KUKA KRL program: EPS_2_251719_MHBURNETSTREET_A_20251210010854.src

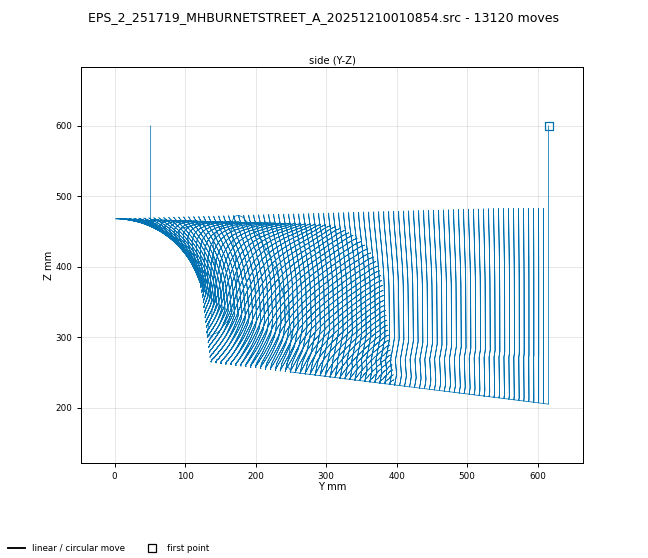
[picture p0: tool path of EPS_2_251719_MHBURNETSTREET_A_20251210010854.src, 13120 of 13122 moves have a stored position in this frame; points joined in program order, loops and branches not executed]
&ACCESS RVP
&REL 4
&COMMENT QRS 19112012
&PARAM EDITMASK = *
DEF PART()
EXT BAS (BAS_COMMAND :IN,REAL :IN )
INT I
BAS (#INITMOV,0 )

;KUKA QRS Post kuka4.cps  Date:22-06-2017 !

File_ID=2951

QRS_PRE_INIT()

;Init var - Until changes are made in qrs_pre_init
Outlet_Square_prg=0
Inlet_1_Square_prg=0
Inlet_2_Square_prg=0
Inlet_3_Square_prg=0
Inlet_4_Square_prg=0
Inlet_5_Square_prg=0

Outlet_1={X 0.000, Y 540.910, Z 382.500, B 0.000, E1 0.000 }
Inlet_1={X 0.000, Y 561.820, Z 357.500, B 0.000, E1 180.000 }
Outlet_1_type=201
Inlet_1_type=0
;QRS#1=Sidecore dimensions
;QRS#2=200-8" PVC SDR 35
;QRS#3=DeadEnd 201
;QRS#4=
;QRS#5=
;QRS#6=
;QRS#7=
;QRS#8=
;QRS#9=12-08 PSX
;QRS#10=

;QRS#11=
;QRS#12=
;QRS#13=
;QRS#14=
;QRS#15=
;QRS#16=1220x127x762 2,5'
;QRS#17=EPS Height
;QRS#18=483
;QRS#19=*
;QRS#20= UPDATED VERSION 22-06-2017
;QRS#21=*
Outlet_Square=0100
Inlet_1_Square=00
Inlet_2_Square=0
Inlet_3_Square=0
Inlet_4_Square=0
Inlet_5_Square=0
Mill_Square=1
Outlet_Square_Prg=204
Inlet_1_Square_prg=0

QRS_INIT()

$ADVANCE=5

; T1
PTP {E1 173.606,E2 173.606}
PTP {X 0,Y 615.507,A -85,B 0,C 180,E1 173.606,E2 173.606,E3 0,E4 0,E5 0,E6 0}
QRS_SPEED_INIT()
LIN {X 0,Y 615.507,Z 600,A -85,B 0,C 180,E1 173.606,E2 173.606,E3 0,E4 0,E5 0,E6 0} C_VEL
LIN {X 0,Y 615.507,Z 215.37,A -85,B 0,C 180,E1 173.606,E2 173.606} C_VEL
LIN {X 0,Y 615.507,Z 207.199,A -85,B 0,C 180,E1 173.606,E2 173.606} C_VEL
LIN {X 0,Y 615.488,Z 205.199,A -85,B 0,C 180,E1 173.42,E2 173.42} C_VEL
LIN {X 0,Y 615.469,Z 205.19,A -85,B 0,C 180,E1 170.801,E2 170.801} C_VEL
LIN {X 0,Y 615.485,Z 205.185,A -85,B 0,C 180,E1 168.14,E2 168.14} C_VEL
LIN {X 0,Y 615.491,Z 205.201,A -85,B 0,C 180,E1 165.451,E2 165.451} C_VEL
LIN {X 0,Y 615.475,Z 205.186,A -85,B 0,C 180,E1 162.73,E2 162.73} C_VEL
LIN {X 0,Y 615.483,Z 205.192,A -85,B 0,C 180,E1 159.968,E2 159.968} C_VEL
LIN {X 0,Y 615.471,Z 205.191,A -85,B 0,C 180,E1 157.155,E2 157.155} C_VEL
LIN {X 0,Y 615.491,Z 205.183,A -85,B 0,C 180,E1 154.43,E2 154.43} C_VEL
LIN {X 0,Y 615.48,Z 205.197,A -85,B 0,C 180,E1 151.551,E2 151.551} C_VEL
LIN {X 0,Y 615.482,Z 205.184,A -85,B 0,C 180,E1 148.915,E2 148.915} C_VEL
LIN {X 0,Y 615.493,Z 205.198,A -85,B 0,C 180,E1 145.979,E2 145.979} C_VEL
LIN {X 0,Y 615.481,Z 205.184,A -85,B 0,C 180,E1 143.064,E2 143.064} C_VEL
LIN {X 0,Y 615.482,Z 205.195,A -85,B 0,C 180,E1 140.25,E2 140.25} C_VEL
LIN {X 0,Y 615.475,Z 205.193,A -85,B 0,C 180,E1 137.647,E2 137.647} C_VEL
LIN {X 0,Y 615.495,Z 205.181,A -85,B 0,C 180,E1 134.933,E2 134.933} C_VEL
LIN {X 0,Y 615.493,Z 205.199,A -85,B 0,C 180,E1 132.081,E2 132.081} C_VEL
LIN {X 0,Y 615.473,Z 205.192,A -85,B 0,C 180,E1 129.751,E2 129.751} C_VEL
LIN {X 0,Y 615.485,Z 205.185,A -85,B 0,C 180,E1 126.937,E2 126.937} C_VEL
LIN {X 0,Y 615.48,Z 205.195,A -85,B 0,C 180,E1 124.022,E2 124.022} C_VEL
LIN {X 0,Y 615.474,Z 205.188,A -85,B 0,C 180,E1 121.686,E2 121.686} C_VEL
LIN {X 0,Y 615.487,Z 205.183,A -85,B 0,C 180,E1 119.406,E2 119.406} C_VEL
LIN {X 0,Y 615.49,Z 205.201,A -85,B 0,C 180,E1 116.444,E2 116.444} C_VEL
LIN {X 0,Y 615.486,Z 205.183,A -85,B 0,C 180,E1 113.556,E2 113.556} C_VEL
LIN {X 0,Y 615.485,Z 205.198,A -85,B 0,C 180,E1 110.731,E2 110.731} C_VEL
LIN {X 0,Y 615.478,Z 205.187,A -85,B 0,C 180,E1 107.957,E2 107.957} C_VEL
LIN {X 0,Y 615.479,Z 205.189,A -85,B 0,C 180,E1 105.226,E2 105.226} C_VEL
LIN {X 0,Y 615.484,Z 205.196,A -85,B 0,C 180,E1 102.53,E2 102.53} C_VEL
LIN {X 0,Y 615.493,Z 205.181,A -85,B 0,C 180,E1 99.862,E2 99.862} C_VEL
LIN {X 0,Y 615.48,Z 205.193,A -85,B 0,C 180,E1 97.216,E2 97.216} C_VEL
LIN {X 0,Y 615.48,Z 205.194,A -85,B 0,C 180,E1 94.585,E2 94.585} C_VEL
LIN {X 0,Y 615.5,Z 205.18,A -85,B 0,C 180,E1 91.963,E2 91.963} C_VEL
LIN {X 0,Y 615.48,Z 205.193,A -85,B 0,C 180,E1 89.346,E2 89.346} C_VEL
LIN {X 0,Y 615.48,Z 205.193,A -85,B 0,C 180,E1 86.727,E2 86.727} C_VEL
LIN {X 0,Y 615.498,Z 205.18,A -85,B 0,C 180,E1 84.102,E2 84.102} C_VEL
LIN {X 0,Y 615.481,Z 205.194,A -85,B 0,C 180,E1 81.463,E2 81.463} C_VEL
LIN {X 0,Y 615.477,Z 205.192,A -85,B 0,C 180,E1 78.807,E2 78.807} C_VEL
LIN {X 0,Y 615.483,Z 205.184,A -85,B 0,C 180,E1 76.067,E2 76.067} C_VEL
LIN {X 0,Y 615.493,Z 205.199,A -85,B 0,C 180,E1 73.414,E2 73.414} C_VEL
LIN {X 0,Y 615.485,Z 205.185,A -85,B 0,C 180,E1 70.662,E2 70.662} C_VEL
LIN {X 0,Y 615.477,Z 205.192,A -85,B 0,C 180,E1 67.863,E2 67.863} C_VEL
LIN {X 0,Y 615.48,Z 205.19,A -85,B 0,C 180,E1 65.008,E2 65.008} C_VEL
LIN {X 0,Y 615.484,Z 205.185,A -85,B 0,C 180,E1 62.823,E2 62.823} C_VEL
LIN {X 0,Y 615.475,Z 205.188,A -85,B 0,C 180,E1 60.206,E2 60.206} C_VEL
LIN {X 0,Y 615.492,Z 205.198,A -85,B 0,C 180,E1 57.543,E2 57.543} C_VEL
LIN {X 0,Y 615.481,Z 205.189,A -85,B 0,C 180,E1 55.185,E2 55.185} C_VEL
LIN {X 0,Y 615.492,Z 205.182,A -85,B 0,C 180,E1 52.758,E2 52.758} C_VEL
LIN {X 0,Y 615.491,Z 205.198,A -85,B 0,C 180,E1 49.91,E2 49.91} C_VEL
LIN {X 0,Y 615.488,Z 205.183,A -85,B 0,C 180,E1 46.952,E2 46.952} C_VEL
LIN {X 0,Y 615.482,Z 205.196,A -85,B 0,C 180,E1 44.149,E2 44.149} C_VEL
LIN {X 0,Y 615.482,Z 205.189,A -85,B 0,C 180,E1 41.474,E2 41.474} C_VEL
LIN {X 0,Y 615.482,Z 205.184,A -85,B 0,C 180,E1 38.904,E2 38.904} C_VEL
LIN {X 0,Y 615.476,Z 205.194,A -85,B 0,C 180,E1 36.425,E2 36.425} C_VEL
LIN {X 0,Y 615.485,Z 205.186,A -85,B 0,C 180,E1 33.534,E2 33.534} C_VEL
LIN {X 0,Y 615.474,Z 205.187,A -85,B 0,C 180,E1 30.92,E2 30.92} C_VEL
LIN {X 0,Y 615.48,Z 205.197,A -85,B 0,C 180,E1 28.449,E2 28.449} C_VEL
LIN {X 0,Y 615.487,Z 205.184,A -85,B 0,C 180,E1 25.569,E2 25.569} C_VEL
LIN {X 0,Y 615.471,Z 205.191,A -85,B 0,C 180,E1 22.845,E2 22.845} C_VEL
LIN {X 0,Y 615.486,Z 205.197,A -85,B 0,C 180,E1 20.557,E2 20.557} C_VEL
LIN {X 0,Y 615.484,Z 205.189,A -85,B 0,C 180,E1 17.957,E2 17.957} C_VEL
LIN {X 0,Y 615.472,Z 205.188,A -85,B 0,C 180,E1 15.226,E2 15.226} C_VEL
LIN {X 0,Y 615.489,Z 205.202,A -85,B 0,C 180,E1 12.53,E2 12.53} C_VEL
LIN {X 0,Y 615.495,Z 205.182,A -85,B 0,C 180,E1 9.862,E2 9.862} C_VEL
LIN {X 0,Y 615.469,Z 205.191,A -85,B 0,C 180,E1 7.215,E2 7.215} C_VEL
LIN {X 0,Y 615.492,Z 205.197,A -85,B 0,C 180,E1 4.584,E2 4.584} C_VEL
LIN {X 0,Y 615.5,Z 205.181,A -85,B 0,C 180,E1 1.963,E2 1.963} C_VEL
LIN {X 0,Y 615.468,Z 205.191,A -85,B 0,C 180,E1 -0.655,E2 -0.655} C_VEL
LIN {X 0,Y 615.492,Z 205.197,A -85,B 0,C 180,E1 -3.273,E2 -3.273} C_VEL
LIN {X 0,Y 615.497,Z 205.181,A -85,B 0,C 180,E1 -5.899,E2 -5.899} C_VEL
LIN {X 0,Y 615.468,Z 205.192,A -85,B 0,C 180,E1 -8.537,E2 -8.537} C_VEL
LIN {X 0,Y 615.489,Z 205.195,A -85,B 0,C 180,E1 -11.193,E2 -11.193} C_VEL
LIN {X 0,Y 615.479,Z 205.184,A -85,B 0,C 180,E1 -13.93,E2 -13.93} C_VEL
LIN {X 0,Y 615.476,Z 205.196,A -85,B 0,C 180,E1 -16.587,E2 -16.587} C_VEL
LIN {X 0,Y 615.489,Z 205.187,A -85,B 0,C 180,E1 -19.338,E2 -19.338} C_VEL
LIN {X 0,Y 615.465,Z 205.191,A -85,B 0,C 180,E1 -22.138,E2 -22.138} C_VEL
LIN {X 0,Y 615.488,Z 205.193,A -85,B 0,C 180,E1 -24.992,E2 -24.992} C_VEL
LIN {X 0,Y 615.466,Z 205.189,A -85,B 0,C 180,E1 -27.916,E2 -27.916} C_VEL
LIN {X 0,Y 615.468,Z 205.194,A -85,B 0,C 180,E1 -30.161,E2 -30.161} C_VEL
LIN {X 0,Y 615.487,Z 205.2,A -85,B 0,C 180,E1 -32.458,E2 -32.458} C_VEL
LIN {X 0,Y 615.488,Z 205.192,A -85,B 0,C 180,E1 -34.815,E2 -34.815} C_VEL
LIN {X 0,Y 615.49,Z 205.183,A -85,B 0,C 180,E1 -37.242,E2 -37.242} C_VEL
LIN {X 0,Y 615.472,Z 205.196,A -85,B 0,C 180,E1 -40.088,E2 -40.088} C_VEL
LIN {X 0,Y 615.488,Z 205.184,A -85,B 0,C 180,E1 -43.048,E2 -43.048} C_VEL
LIN {X 0,Y 615.467,Z 205.194,A -85,B 0,C 180,E1 -45.849,E2 -45.849} C_VEL
LIN {X 0,Y 615.489,Z 205.192,A -85,B 0,C 180,E1 -48.527,E2 -48.527} C_VEL
LIN {X 0,Y 615.478,Z 205.185,A -85,B 0,C 180,E1 -51.095,E2 -51.095} C_VEL
LIN {X 0,Y 615.463,Z 205.192,A -85,B 0,C 180,E1 -53.574,E2 -53.574} C_VEL
LIN {X 0,Y 615.49,Z 205.189,A -85,B 0,C 180,E1 -56.466,E2 -56.466} C_VEL
LIN {X 0,Y 615.467,Z 205.187,A -85,B 0,C 180,E1 -59.079,E2 -59.079} C_VEL
LIN {X 0,Y 615.466,Z 205.195,A -85,B 0,C 180,E1 -61.554,E2 -61.554} C_VEL
LIN {X 0,Y 615.49,Z 205.187,A -85,B 0,C 180,E1 -64.431,E2 -64.431} C_VEL
LIN {X 0,Y 615.497,Z 205.361,A -85,B 0,C 180,E1 -65.958,E2 -65.958} C_VEL
LIN {X 0,Y 615.49,Z 220.439,A -85,B 0,C 180,E1 -68.568,E2 -68.568} C_VEL
LIN {X 0,Y 615.483,Z 237.22,A -85,B 0,C 180,E1 -71.397,E2 -71.397} C_VEL
LIN {X 0,Y 615.498,Z 254.497,A -85,B 0,C 180,E1 -74.265,E2 -74.265} C_VEL
LIN {X 0,Y 615.469,Z 271.731,A -85,B 0,C 180,E1 -77.071,E2 -77.071} C_VEL
LIN {X 0,Y 615.463,Z 273.25,A -85,B 0,C 180,E1 -77.155,E2 -77.155} C_VEL
LIN {X 0,Y 615.498,Z 378.83,A -85,B 0,C 180,E1 -78.411,E2 -78.411} C_VEL
LIN {X 0,Y 615.499,Z 391.343,A -85,B 0,C 180,E1 -78.682,E2 -78.682} C_VEL
LIN {X 0,Y 615.496,Z 404.502,A -85,B 0,C 180,E1 -79.109,E2 -79.109} C_VEL
LIN {X 0,Y 615.488,Z 416.478,A -85,B 0,C 180,E1 -79.639,E2 -79.639} C_VEL
LIN {X 0,Y 615.494,Z 427.994,A -85,B 0,C 180,E1 -80.304,E2 -80.304} C_VEL
LIN {X 0,Y 615.499,Z 438.341,A -85,B 0,C 180,E1 -81.05,E2 -81.05} C_VEL
LIN {X 0,Y 615.497,Z 446.812,A -85,B 0,C 180,E1 -81.794,E2 -81.794} C_VEL
LIN {X 0,Y 615.498,Z 454.606,A -85,B 0,C 180,E1 -82.62,E2 -82.62} C_VEL
LIN {X 0,Y 615.496,Z 462.203,A -85,B 0,C 180,E1 -83.608,E2 -83.608} C_VEL
LIN {X 0,Y 615.498,Z 469.205,A -85,B 0,C 180,E1 -84.759,E2 -84.759} C_VEL
LIN {X 0,Y 615.494,Z 473.851,A -85,B 0,C 180,E1 -85.744,E2 -85.744} C_VEL
LIN {X 0,Y 615.494,Z 477.399,A -85,B 0,C 180,E1 -86.727,E2 -86.727} C_VEL
LIN {X 0,Y 615.497,Z 479.233,A -85,B 0,C 180,E1 -87.382,E2 -87.382} C_VEL
LIN {X 0,Y 615.5,Z 480.607,A -85,B 0,C 180,E1 -88.037,E2 -88.037} C_VEL
LIN {X 0,Y 615.496,Z 482.173,A -85,B 0,C 180,E1 -89.346,E2 -89.346} C_VEL
LIN {X 0,Y 615.494,Z 482.389,A -85,B 0,C 180,E1 -90,E2 -90} C_VEL
LIN {X 0,Y 615.495,Z 481.58,A -85,B 0,C 180,E1 -91.309,E2 -91.309} C_VEL
LIN {X 0,Y 615.5,Z 480.607,A -85,B 0,C 180,E1 -91.963,E2 -91.963} C_VEL
LIN {X 0,Y 615.497,Z 479.233,A -85,B 0,C 180,E1 -92.618,E2 -92.618} C_VEL
LIN {X 0,Y 615.496,Z 476.349,A -85,B 0,C 180,E1 -93.601,E2 -93.601} C_VEL
LIN {X 0,Y 615.498,Z 472.441,A -85,B 0,C 180,E1 -94.584,E2 -94.584} C_VEL
LIN {X 0,Y 615.499,Z 467.405,A -85,B 0,C 180,E1 -95.57,E2 -95.57} C_VEL
LIN {X 0,Y 615.497,Z 460.87,A -85,B 0,C 180,E1 -96.583,E2 -96.583} C_VEL
LIN {X 0,Y 615.497,Z 453.133,A -85,B 0,C 180,E1 -97.545,E2 -97.545} C_VEL
LIN {X 0,Y 615.498,Z 445.045,A -85,B 0,C 180,E1 -98.371,E2 -98.371} C_VEL
LIN {X 0,Y 615.499,Z 435.168,A -85,B 0,C 180,E1 -99.199,E2 -99.199} C_VEL
LIN {X 0,Y 615.491,Z 423.982,A -85,B 0,C 180,E1 -99.945,E2 -99.945} C_VEL
LIN {X 0,Y 615.493,Z 413.022,A -85,B 0,C 180,E1 -100.527,E2 -100.527} C_VEL
LIN {X 0,Y 615.499,Z 400.419,A -85,B 0,C 180,E1 -101.042,E2 -101.042} C_VEL
LIN {X 0,Y 615.499,Z 388.065,A -85,B 0,C 180,E1 -101.401,E2 -101.401} C_VEL
LIN {X 0,Y 615.499,Z 374.466,A -85,B 0,C 180,E1 -101.652,E2 -101.652} C_VEL
LIN {X 0,Y 615.465,Z 272.546,A -85,B 0,C 180,E1 -102.866,E2 -102.866} C_VEL
LIN {X 0,Y 615.478,Z 270.987,A -85,B 0,C 180,E1 -103.033,E2 -103.033} C_VEL
LIN {X 0,Y 615.494,Z 253.464,A -85,B 0,C 180,E1 -105.905,E2 -105.905} C_VEL
LIN {X 0,Y 615.484,Z 236.96,A -85,B 0,C 180,E1 -108.646,E2 -108.646} C_VEL
LIN {X 0,Y 615.49,Z 220.439,A -85,B 0,C 180,E1 -111.432,E2 -111.432} C_VEL
LIN {X 0,Y 615.497,Z 205.361,A -85,B 0,C 180,E1 -114.042,E2 -114.042} C_VEL
LIN {X 0,Y 615.468,Z 205.195,A -85,B 0,C 180,E1 -116.445,E2 -116.445} C_VEL
LIN {X 0,Y 615.461,Z 205.192,A -85,B 0,C 180,E1 -118.659,E2 -118.659} C_VEL
LIN {X 0,Y 615.478,Z 205.185,A -85,B 0,C 180,E1 -121.084,E2 -121.084} C_VEL
LIN {X 0,Y 615.486,Z 205.2,A -85,B 0,C 180,E1 -124.022,E2 -124.022} C_VEL
LIN {X 0,Y 615.463,Z 205.192,A -85,B 0,C 180,E1 -126.426,E2 -126.426} C_VEL
LIN {X 0,Y 615.493,Z 205.183,A -85,B 0,C 180,E1 -129.062,E2 -129.062} C_VEL
LIN {X 0,Y 615.472,Z 205.196,A -85,B 0,C 180,E1 -132.078,E2 -132.078} C_VEL
LIN {X 0,Y 615.493,Z 205.182,A -85,B 0,C 180,E1 -134.932,E2 -134.932} C_VEL
LIN {X 0,Y 615.475,Z 205.196,A -85,B 0,C 180,E1 -137.921,E2 -137.921} C_VEL
LIN {X 0,Y 615.462,Z 205.191,A -85,B 0,C 180,E1 -140.248,E2 -140.248} C_VEL
LIN {X 0,Y 615.49,Z 205.188,A -85,B 0,C 180,E1 -143.063,E2 -143.063} C_VEL
LIN {X 0,Y 615.466,Z 205.193,A -85,B 0,C 180,E1 -145.976,E2 -145.976} C_VEL
LIN {X 0,Y 615.467,Z 205.188,A -85,B 0,C 180,E1 -148.313,E2 -148.313} C_VEL
LIN {X 0,Y 615.486,Z 205.184,A -85,B 0,C 180,E1 -150.593,E2 -150.593} C_VEL
LIN {X 0,Y 615.478,Z 205.197,A -85,B 0,C 180,E1 -153.555,E2 -153.555} C_VEL
LIN {X 0,Y 615.465,Z 205.189,A -85,B 0,C 180,E1 -155.996,E2 -155.996} C_VEL
LIN {X 0,Y 615.495,Z 205.183,A -85,B 0,C 180,E1 -158.568,E2 -158.568} C_VEL
LIN {X 0,Y 615.479,Z 205.197,A -85,B 0,C 180,E1 -161.397,E2 -161.397} C_VEL
LIN {X 0,Y 615.478,Z 205.185,A -85,B 0,C 180,E1 -164.094,E2 -164.094} C_VEL
LIN {X 0,Y 615.486,Z 205.194,A -85,B 0,C 180,E1 -166.798,E2 -166.798} C_VEL
LIN {X 0,Y 615.469,Z 205.193,A -85,B 0,C 180,E1 -169.472,E2 -169.472} C_VEL
LIN {X 0,Y 615.485,Z 205.184,A -85,B 0,C 180,E1 -172.124,E2 -172.124} C_VEL
LIN {X 0,Y 615.489,Z 205.197,A -85,B 0,C 180,E1 -174.758,E2 -174.758} C_VEL
LIN {X 0,Y 615.465,Z 205.192,A -85,B 0,C 180,E1 -177.382,E2 -177.382} C_VEL
LIN {X 0,Y 615.486,Z 205.184,A -85,B 0,C 180,E1 -180,E2 -180} C_VEL
LIN {X 0,Y 615.488,Z 205.198,A -85,B 0,C 180,E1 -182.617,E2 -182.617} C_VEL
LIN {X 0,Y 615.468,Z 205.191,A -85,B 0,C 180,E1 -185.241,E2 -185.241} C_VEL
LIN {X 0,Y 615.488,Z 205.199,A -85,B 0,C 180,E1 -186.58,E2 -186.58} C_VEL
LIN {X 0,Y 614.798,Z 205.338,A -85,B 0,C 180,E1 -187.126,E2 -187.126} C_VEL
LIN {X 0,Y 611.952,Z 205.753,A -85,B 0,C 180,E1 -188.012,E2 -188.012} C_VEL
LIN {X 0,Y 609.562,Z 206.062,A -85,B 0,C 180,E1 -188.725,E2 -188.725} C_VEL
LIN {X 0,Y 608.536,Z 206.179,A -85,B 0,C 180,E1 -189.274,E2 -189.274} C_VEL
LIN {X 0,Y 608.452,Z 206.187,A -85,B 0,C 180,E1 -189.46,E2 -189.46} C_VEL
LIN {X 0,Y 608.462,Z 206.188,A -85,B 0,C 180,E1 -191.999,E2 -191.999} C_VEL
LIN {X 0,Y 608.474,Z 206.192,A -85,B 0,C 180,E1 -194.72,E2 -194.72} C_VEL
LIN {X 0,Y 608.445,Z 206.188,A -85,B 0,C 180,E1 -197.476,E2 -197.476} C_VEL
LIN {X 0,Y 608.461,Z 206.194,A -85,B 0,C 180,E1 -200.274,E2 -200.274} C_VEL
LIN {X 0,Y 608.456,Z 206.196,A -85,B 0,C 180,E1 -202.476,E2 -202.476} C_VEL
LIN {X 0,Y 608.449,Z 206.194,A -85,B 0,C 180,E1 -204.571,E2 -204.571} C_VEL
LIN {X 0,Y 608.473,Z 206.185,A -85,B 0,C 180,E1 -207.207,E2 -207.207} C_VEL
LIN {X 0,Y 608.469,Z 206.192,A -85,B 0,C 180,E1 -209.972,E2 -209.972} C_VEL
LIN {X 0,Y 608.454,Z 206.192,A -85,B 0,C 180,E1 -212.522,E2 -212.522} C_VEL
LIN {X 0,Y 608.44,Z 206.189,A -85,B 0,C 180,E1 -214.905,E2 -214.905} C_VEL
LIN {X 0,Y 608.479,Z 206.184,A -85,B 0,C 180,E1 -217.16,E2 -217.16} C_VEL
LIN {X 0,Y 608.474,Z 206.187,A -85,B 0,C 180,E1 -219.439,E2 -219.439} C_VEL
LIN {X 0,Y 608.447,Z 206.192,A -85,B 0,C 180,E1 -222.333,E2 -222.333} C_VEL
LIN {X 0,Y 608.46,Z 206.187,A -85,B 0,C 180,E1 -224.795,E2 -224.795} C_VEL
LIN {X 0,Y 608.454,Z 206.187,A -85,B 0,C 180,E1 -227.04,E2 -227.04} C_VEL
LIN {X 0,Y 608.453,Z 206.196,A -85,B 0,C 180,E1 -229.697,E2 -229.697} C_VEL
LIN {X 0,Y 608.469,Z 206.188,A -85,B 0,C 180,E1 -232.254,E2 -232.254} C_VEL
LIN {X 0,Y 608.445,Z 206.19,A -85,B 0,C 180,E1 -235.094,E2 -235.094} C_VEL
LIN {X 0,Y 608.467,Z 206.192,A -85,B 0,C 180,E1 -237.906,E2 -237.906} C_VEL
LIN {X 0,Y 608.46,Z 206.188,A -85,B 0,C 180,E1 -240.22,E2 -240.22} C_VEL
LIN {X 0,Y 608.477,Z 206.185,A -85,B 0,C 180,E1 -242.792,E2 -242.792} C_VEL
LIN {X 0,Y 608.449,Z 206.198,A -85,B 0,C 180,E1 -245.429,E2 -245.429} C_VEL
LIN {X 0,Y 608.469,Z 206.186,A -85,B 0,C 180,E1 -248.309,E2 -248.309} C_VEL
LIN {X 0,Y 608.472,Z 206.194,A -85,B 0,C 180,E1 -251.282,E2 -251.282} C_VEL
LIN {X 0,Y 608.457,Z 206.189,A -85,B 0,C 180,E1 -253.906,E2 -253.906} C_VEL
LIN {X 0,Y 608.459,Z 206.188,A -85,B 0,C 180,E1 -256.644,E2 -256.644} C_VEL
LIN {X 0,Y 608.463,Z 206.194,A -85,B 0,C 180,E1 -259.35,E2 -259.35} C_VEL
LIN {X 0,Y 608.477,Z 206.185,A -85,B 0,C 180,E1 -262.033,E2 -262.033} C_VEL
LIN {X 0,Y 608.461,Z 206.19,A -85,B 0,C 180,E1 -264.698,E2 -264.698} C_VEL
LIN {X 0,Y 608.472,Z 206.191,A -85,B 0,C 180,E1 -267.352,E2 -267.352} C_VEL
LIN {X 0,Y 608.477,Z 206.185,A -85,B 0,C 180,E1 -270,E2 -270} C_VEL
LIN {X 0,Y 608.472,Z 206.191,A -85,B 0,C 180,E1 -272.648,E2 -272.648} C_VEL
LIN {X 0,Y 608.461,Z 206.19,A -85,B 0,C 180,E1 -275.302,E2 -275.302} C_VEL
LIN {X 0,Y 608.477,Z 206.185,A -85,B 0,C 180,E1 -277.967,E2 -277.967} C_VEL
LIN {X 0,Y 608.468,Z 206.193,A -85,B 0,C 180,E1 -280.958,E2 -280.958} C_VEL
LIN {X 0,Y 608.459,Z 206.188,A -85,B 0,C 180,E1 -283.356,E2 -283.356} C_VEL
LIN {X 0,Y 608.457,Z 206.189,A -85,B 0,C 180,E1 -286.094,E2 -286.094} C_VEL
LIN {X 0,Y 608.456,Z 206.193,A -85,B 0,C 180,E1 -288.87,E2 -288.87} C_VEL
LIN {X 0,Y 608.469,Z 206.186,A -85,B 0,C 180,E1 -291.691,E2 -291.691} C_VEL
LIN {X 0,Y 608.449,Z 206.198,A -85,B 0,C 180,E1 -294.571,E2 -294.571} C_VEL
LIN {X 0,Y 608.477,Z 206.185,A -85,B 0,C 180,E1 -297.208,E2 -297.208} C_VEL
LIN {X 0,Y 608.458,Z 206.19,A -85,B 0,C 180,E1 -299.971,E2 -299.971} C_VEL
LIN {X 0,Y 608.466,Z 206.193,A -85,B 0,C 180,E1 -302.524,E2 -302.524} C_VEL
LIN {X 0,Y 608.435,Z 206.189,A -85,B 0,C 180,E1 -305.278,E2 -305.278} C_VEL
LIN {X 0,Y 608.469,Z 206.188,A -85,B 0,C 180,E1 -307.746,E2 -307.746} C_VEL
LIN {X 0,Y 608.452,Z 206.195,A -85,B 0,C 180,E1 -310.33,E2 -310.33} C_VEL
LIN {X 0,Y 608.454,Z 206.187,A -85,B 0,C 180,E1 -312.96,E2 -312.96} C_VEL
LIN {X 0,Y 608.453,Z 206.192,A -85,B 0,C 180,E1 -315.736,E2 -315.736} C_VEL
LIN {X 0,Y 608.46,Z 206.188,A -85,B 0,C 180,E1 -318.658,E2 -318.658} C_VEL
LIN {X 0,Y 608.466,Z 206.188,A -85,B 0,C 180,E1 -321.412,E2 -321.412} C_VEL
LIN {X 0,Y 608.474,Z 206.195,A -85,B 0,C 180,E1 -323.951,E2 -323.951} C_VEL
LIN {X 0,Y 608.465,Z 206.189,A -85,B 0,C 180,E1 -326.33,E2 -326.33} C_VEL
LIN {X 0,Y 608.474,Z 206.185,A -85,B 0,C 180,E1 -328.728,E2 -328.728} C_VEL
LIN {X 0,Y 608.464,Z 206.19,A -85,B 0,C 180,E1 -331.381,E2 -331.381} C_VEL
LIN {X 0,Y 608.443,Z 206.195,A -85,B 0,C 180,E1 -333.965,E2 -333.965} C_VEL
LIN {X 0,Y 608.466,Z 206.189,A -85,B 0,C 180,E1 -336.156,E2 -336.156} C_VEL
LIN {X 0,Y 608.472,Z 206.186,A -85,B 0,C 180,E1 -338.309,E2 -338.309} C_VEL
LIN {X 0,Y 608.468,Z 206.191,A -85,B 0,C 180,E1 -341.284,E2 -341.284} C_VEL
LIN {X 0,Y 608.462,Z 206.19,A -85,B 0,C 180,E1 -343.907,E2 -343.907} C_VEL
LIN {X 0,Y 608.453,Z 206.188,A -85,B 0,C 180,E1 -346.644,E2 -346.644} C_VEL
LIN {X 0,Y 608.463,Z 206.196,A -85,B 0,C 180,E1 -349.351,E2 -349.351} C_VEL
LIN {X 0,Y 608.479,Z 206.185,A -85,B 0,C 180,E1 -352.033,E2 -352.033} C_VEL
LIN {X 0,Y 608.45,Z 206.189,A -85,B 0,C 180,E1 -354.698,E2 -354.698} C_VEL
LIN {X 0,Y 608.478,Z 206.193,A -85,B 0,C 180,E1 -357.352,E2 -357.352} C_VEL
LIN {X 0,Y 608.477,Z 206.184,A -85,B 0,C 180,E1 -360,E2 -360} C_VEL
LIN {X 0,Y 608.459,Z 206.189,A -85,B 0,C 180,E1 -362.648,E2 -362.648} C_VEL
LIN {X 0,Y 608.469,Z 206.192,A -85,B 0,C 180,E1 -365.302,E2 -365.302} C_VEL
LIN {X 0,Y 608.475,Z 206.184,A -85,B 0,C 180,E1 -367.967,E2 -367.967} C_VEL
LIN {X 0,Y 608.453,Z 206.192,A -85,B 0,C 180,E1 -370.65,E2 -370.65} C_VEL
LIN {X 0,Y 608.463,Z 206.19,A -85,B 0,C 180,E1 -373.357,E2 -373.357} C_VEL
LIN {X 0,Y 608.45,Z 206.188,A -85,B 0,C 180,E1 -376.094,E2 -376.094} C_VEL
LIN {X 0,Y 608.453,Z 206.197,A -85,B 0,C 180,E1 -378.87,E2 -378.87} C_VEL
LIN {X 0,Y 608.466,Z 206.186,A -85,B 0,C 180,E1 -381.692,E2 -381.692} C_VEL
LIN {X 0,Y 608.445,Z 206.197,A -85,B 0,C 180,E1 -384.572,E2 -384.572} C_VEL
LIN {X 0,Y 608.481,Z 206.186,A -85,B 0,C 180,E1 -387.208,E2 -387.208} C_VEL
LIN {X 0,Y 608.451,Z 206.189,A -85,B 0,C 180,E1 -389.969,E2 -389.969} C_VEL
LIN {X 0,Y 608.459,Z 206.191,A -85,B 0,C 180,E1 -392.88,E2 -392.88} C_VEL
LIN {X 0,Y 608.435,Z 206.19,A -85,B 0,C 180,E1 -395.279,E2 -395.279} C_VEL
LIN {X 0,Y 608.459,Z 206.188,A -85,B 0,C 180,E1 -397.747,E2 -397.747} C_VEL
LIN {X 0,Y 608.446,Z 206.198,A -85,B 0,C 180,E1 -400.329,E2 -400.329} C_VEL
LIN {X 0,Y 608.469,Z 206.185,A -85,B 0,C 180,E1 -403.309,E2 -403.309} C_VEL
LIN {X 0,Y 608.463,Z 206.194,A -85,B 0,C 180,E1 -406.13,E2 -406.13} C_VEL
LIN {X 0,Y 608.457,Z 206.188,A -85,B 0,C 180,E1 -408.824,E2 -408.824} C_VEL
LIN {X 0,Y 608.433,Z 206.19,A -85,B 0,C 180,E1 -411.41,E2 -411.41} C_VEL
LIN {X 0,Y 608.448,Z 206.196,A -85,B 0,C 180,E1 -413.955,E2 -413.955} C_VEL
LIN {X 0,Y 608.466,Z 206.192,A -85,B 0,C 180,E1 -416.33,E2 -416.33} C_VEL
LIN {X 0,Y 608.447,Z 206.189,A -85,B 0,C 180,E1 -418.733,E2 -418.733} C_VEL
LIN {X 0,Y 608.454,Z 206.189,A -85,B 0,C 180,E1 -421.384,E2 -421.384} C_VEL
LIN {X 0,Y 608.439,Z 206.2,A -85,B 0,C 180,E1 -423.964,E2 -423.964} C_VEL
LIN {X 0,Y 608.496,Z 206.349,A -85,B 0,C 180,E1 -425.844,E2 -425.844} C_VEL
LIN {X 0,Y 608.529,Z 220.462,A -85,B 0,C 180,E1 -428.311,E2 -428.311} C_VEL
LIN {X 0,Y 608.51,Z 237.019,A -85,B 0,C 180,E1 -431.132,E2 -431.132} C_VEL
LIN {X 0,Y 608.483,Z 253.576,A -85,B 0,C 180,E1 -433.907,E2 -433.907} C_VEL
LIN {X 0,Y 608.48,Z 270.133,A -85,B 0,C 180,E1 -436.644,E2 -436.644} C_VEL
LIN {X 0,Y 608.461,Z 272.248,A -85,B 0,C 180,E1 -436.962,E2 -436.962} C_VEL
LIN {X 0,Y 608.539,Z 274.724,A -85,B 0,C 180,E1 -437.028,E2 -437.028} C_VEL
LIN {X 0,Y 608.548,Z 378.941,A -85,B 0,C 180,E1 -438.277,E2 -438.277} C_VEL
LIN {X 0,Y 608.548,Z 392.226,A -85,B 0,C 180,E1 -438.572,E2 -438.572} C_VEL
LIN {X 0,Y 608.54,Z 405.391,A -85,B 0,C 180,E1 -439.011,E2 -439.011} C_VEL
LIN {X 0,Y 608.51,Z 416.623,A -85,B 0,C 180,E1 -439.519,E2 -439.519} C_VEL
LIN {X 0,Y 608.485,Z 428.198,A -85,B 0,C 180,E1 -440.191,E2 -440.191} C_VEL
LIN {X 0,Y 608.485,Z 438.596,A -85,B 0,C 180,E1 -440.946,E2 -440.946} C_VEL
LIN {X 0,Y 608.475,Z 447.114,A -85,B 0,C 180,E1 -441.699,E2 -441.699} C_VEL
LIN {X 0,Y 608.471,Z 454.959,A -85,B 0,C 180,E1 -442.534,E2 -442.534} C_VEL
LIN {X 0,Y 608.461,Z 462.286,A -85,B 0,C 180,E1 -443.485,E2 -443.485} C_VEL
LIN {X 0,Y 608.451,Z 467.864,A -85,B 0,C 180,E1 -444.366,E2 -444.366} C_VEL
LIN {X 0,Y 608.432,Z 472.95,A -85,B 0,C 180,E1 -445.362,E2 -445.362} C_VEL
LIN {X 0,Y 608.449,Z 476.896,A -85,B 0,C 180,E1 -446.358,E2 -446.358} C_VEL
LIN {X 0,Y 608.425,Z 479.808,A -85,B 0,C 180,E1 -447.352,E2 -447.352} C_VEL
LIN {X 0,Y 608.445,Z 481.201,A -85,B 0,C 180,E1 -448.014,E2 -448.014} C_VEL
LIN {X 0,Y 608.438,Z 482.783,A -85,B 0,C 180,E1 -449.338,E2 -449.338} C_VEL
LIN {X 0,Y 608.434,Z 482.998,A -85,B 0,C 180,E1 -450,E2 -450} C_VEL
LIN {X 0,Y 608.448,Z 482.184,A -85,B 0,C 180,E1 -451.324,E2 -451.324} C_VEL
LIN {X 0,Y 608.445,Z 481.201,A -85,B 0,C 180,E1 -451.986,E2 -451.986} C_VEL
LIN {X 0,Y 608.425,Z 479.808,A -85,B 0,C 180,E1 -452.648,E2 -452.648} C_VEL
LIN {X 0,Y 608.449,Z 476.896,A -85,B 0,C 180,E1 -453.642,E2 -453.642} C_VEL
LIN {X 0,Y 608.432,Z 472.95,A -85,B 0,C 180,E1 -454.638,E2 -454.638} C_VEL
LIN {X 0,Y 608.451,Z 467.864,A -85,B 0,C 180,E1 -455.634,E2 -455.634} C_VEL
LIN {X 0,Y 608.442,Z 461.472,A -85,B 0,C 180,E1 -456.633,E2 -456.633} C_VEL
LIN {X 0,Y 608.475,Z 453.479,A -85,B 0,C 180,E1 -457.633,E2 -457.633} C_VEL
LIN {X 0,Y 608.487,Z 445.338,A -85,B 0,C 180,E1 -458.468,E2 -458.468} C_VEL
LIN {X 0,Y 608.487,Z 435.396,A -85,B 0,C 180,E1 -459.306,E2 -459.306} C_VEL
LIN {X 0,Y 608.505,Z 424.168,A -85,B 0,C 180,E1 -460.06,E2 -460.06} C_VEL
LIN {X 0,Y 608.518,Z 413.176,A -85,B 0,C 180,E1 -460.649,E2 -460.649} C_VEL
LIN {X 0,Y 608.535,Z 401.706,A -85,B 0,C 180,E1 -461.127,E2 -461.127} C_VEL
LIN {X 0,Y 608.55,Z 389.069,A -85,B 0,C 180,E1 -461.512,E2 -461.512} C_VEL
LIN {X 0,Y 608.563,Z 376.111,A -85,B 0,C 180,E1 -461.765,E2 -461.765} C_VEL
LIN {X 0,Y 608.48,Z 272.577,A -85,B 0,C 180,E1 -463.016,E2 -463.016} C_VEL
LIN {X 0,Y 608.456,Z 271.167,A -85,B 0,C 180,E1 -463.187,E2 -463.187} C_VEL
LIN {X 0,Y 608.498,Z 254.611,A -85,B 0,C 180,E1 -465.921,E2 -465.921} C_VEL
LIN {X 0,Y 608.512,Z 237.855,A -85,B 0,C 180,E1 -468.727,E2 -468.727} C_VEL
LIN {X 0,Y 608.522,Z 222.532,A -85,B 0,C 180,E1 -471.334,E2 -471.334} C_VEL
LIN {X 0,Y 608.552,Z 206.737,A -85,B 0,C 180,E1 -474.072,E2 -474.072} C_VEL
LIN {X 0,Y 608.475,Z 206.255,A -85,B 0,C 180,E1 -474.198,E2 -474.198} C_VEL
LIN {X 0,Y 608.431,Z 206.191,A -85,B 0,C 180,E1 -476.775,E2 -476.775} C_VEL
LIN {X 0,Y 608.476,Z 206.191,A -85,B 0,C 180,E1 -479.779,E2 -479.779} C_VEL
LIN {X 0,Y 608.443,Z 206.191,A -85,B 0,C 180,E1 -482.519,E2 -482.519} C_VEL
LIN {X 0,Y 608.435,Z 206.19,A -85,B 0,C 180,E1 -484.903,E2 -484.903} C_VEL
LIN {X 0,Y 608.468,Z 206.194,A -85,B 0,C 180,E1 -487.746,E2 -487.746} C_VEL
LIN {X 0,Y 608.435,Z 206.192,A -85,B 0,C 180,E1 -490.327,E2 -490.327} C_VEL
LIN {X 0,Y 608.452,Z 206.188,A -85,B 0,C 180,E1 -492.96,E2 -492.96} C_VEL
LIN {X 0,Y 608.455,Z 206.197,A -85,B 0,C 180,E1 -495.736,E2 -495.736} C_VEL
LIN {X 0,Y 608.453,Z 206.187,A -85,B 0,C 180,E1 -498.658,E2 -498.658} C_VEL
LIN {X 0,Y 608.457,Z 206.194,A -85,B 0,C 180,E1 -501.761,E2 -501.761} C_VEL
LIN {X 0,Y 608.441,Z 206.192,A -85,B 0,C 180,E1 -503.955,E2 -503.955} C_VEL
LIN {X 0,Y 608.443,Z 206.189,A -85,B 0,C 180,E1 -506.328,E2 -506.328} C_VEL
LIN {X 0,Y 608.448,Z 206.189,A -85,B 0,C 180,E1 -508.732,E2 -508.732} C_VEL
LIN {X 0,Y 608.472,Z 206.196,A -85,B 0,C 180,E1 -511.38,E2 -511.38} C_VEL
LIN {X 0,Y 608.436,Z 206.191,A -85,B 0,C 180,E1 -513.964,E2 -513.964} C_VEL
LIN {X 0,Y 608.454,Z 206.191,A -85,B 0,C 180,E1 -516.876,E2 -516.876} C_VEL
LIN {X 0,Y 608.463,Z 206.195,A -85,B 0,C 180,E1 -519.322,E2 -519.322} C_VEL
LIN {X 0,Y 608.437,Z 206.19,A -85,B 0,C 180,E1 -521.827,E2 -521.827} C_VEL
LIN {X 0,Y 608.469,Z 206.188,A -85,B 0,C 180,E1 -524.594,E2 -524.594} C_VEL
LIN {X 0,Y 608.464,Z 206.192,A -85,B 0,C 180,E1 -527.322,E2 -527.322} C_VEL
LIN {X 0,Y 608.458,Z 206.186,A -85,B 0,C 180,E1 -530.022,E2 -530.022} C_VEL
LIN {X 0,Y 608.467,Z 206.192,A -85,B 0,C 180,E1 -532.7,E2 -532.7} C_VEL
LIN {X 0,Y 608.469,Z 206.192,A -85,B 0,C 180,E1 -534.698,E2 -534.698} C_VEL
LIN {X 0,Y 608.459,Z 206.189,A -85,B 0,C 180,E1 -537.352,E2 -537.352} C_VEL
LIN {X 0,Y 608.477,Z 206.184,A -85,B 0,C 180,E1 -540,E2 -540} C_VEL
LIN {X 0,Y 608.478,Z 206.193,A -85,B 0,C 180,E1 -542.648,E2 -542.648} C_VEL
LIN {X 0,Y 608.451,Z 206.189,A -85,B 0,C 180,E1 -545.302,E2 -545.302} C_VEL
LIN {X 0,Y 608.479,Z 206.185,A -85,B 0,C 180,E1 -547.967,E2 -547.967} C_VEL
LIN {X 0,Y 608.452,Z 206.187,A -85,B 0,C 180,E1 -549.46,E2 -549.46} C_VEL
LIN {X 0,Y 607.783,Z 206.273,A -85,B 0,C 180,E1 -550.013,E2 -550.013} C_VEL
LIN {X 0,Y 604.933,Z 206.63,A -85,B 0,C 180,E1 -550.91,E2 -550.91} C_VEL
LIN {X 0,Y 602.527,Z 206.929,A -85,B 0,C 180,E1 -551.631,E2 -551.631} C_VEL
LIN {X 0,Y 601.493,Z 207.058,A -85,B 0,C 180,E1 -552.188,E2 -552.188} C_VEL
LIN {X 0,Y 601.408,Z 207.068,A -85,B 0,C 180,E1 -552.376,E2 -552.376} C_VEL
LIN {X 0,Y 601.427,Z 207.067,A -85,B 0,C 180,E1 -554.897,E2 -554.897} C_VEL
LIN {X 0,Y 601.428,Z 207.065,A -85,B 0,C 180,E1 -556.986,E2 -556.986} C_VEL
LIN {X 0,Y 601.403,Z 207.066,A -85,B 0,C 180,E1 -559.809,E2 -559.809} C_VEL
LIN {X 0,Y 601.409,Z 207.07,A -85,B 0,C 180,E1 -562.683,E2 -562.683} C_VEL
LIN {X 0,Y 601.399,Z 207.068,A -85,B 0,C 180,E1 -564.878,E2 -564.878} C_VEL
LIN {X 0,Y 601.412,Z 207.064,A -85,B 0,C 180,E1 -567.362,E2 -567.362} C_VEL
LIN {X 0,Y 601.426,Z 207.073,A -85,B 0,C 180,E1 -570.164,E2 -570.164} C_VEL
LIN {X 0,Y 601.417,Z 207.066,A -85,B 0,C 180,E1 -572.715,E2 -572.715} C_VEL
LIN {X 0,Y 601.389,Z 207.067,A -85,B 0,C 180,E1 -575.111,E2 -575.111} C_VEL
LIN {X 0,Y 601.434,Z 207.063,A -85,B 0,C 180,E1 -577.419,E2 -577.419} C_VEL
LIN {X 0,Y 601.409,Z 207.075,A -85,B 0,C 180,E1 -579.995,E2 -579.995} C_VEL
LIN {X 0,Y 601.408,Z 207.066,A -85,B 0,C 180,E1 -582.67,E2 -582.67} C_VEL
LIN {X 0,Y 601.422,Z 207.067,A -85,B 0,C 180,E1 -585.482,E2 -585.482} C_VEL
LIN {X 0,Y 601.422,Z 207.064,A -85,B 0,C 180,E1 -588.406,E2 -588.406} C_VEL
LIN {X 0,Y 601.435,Z 207.062,A -85,B 0,C 180,E1 -590.875,E2 -590.875} C_VEL
LIN {X 0,Y 601.429,Z 207.072,A -85,B 0,C 180,E1 -593.735,E2 -593.735} C_VEL
LIN {X 0,Y 601.426,Z 207.062,A -85,B 0,C 180,E1 -596.687,E2 -596.687} C_VEL
LIN {X 0,Y 601.427,Z 207.065,A -85,B 0,C 180,E1 -599.059,E2 -599.059} C_VEL
LIN {X 0,Y 601.436,Z 207.068,A -85,B 0,C 180,E1 -601.374,E2 -601.374} C_VEL
LIN {X 0,Y 601.401,Z 207.075,A -85,B 0,C 180,E1 -603.636,E2 -603.636} C_VEL
LIN {X 0,Y 601.416,Z 207.064,A -85,B 0,C 180,E1 -606.59,E2 -606.59} C_VEL
LIN {X 0,Y 601.429,Z 207.072,A -85,B 0,C 180,E1 -609.478,E2 -609.478} C_VEL
LIN {X 0,Y 601.392,Z 207.067,A -85,B 0,C 180,E1 -612.312,E2 -612.312} C_VEL
LIN {X 0,Y 601.41,Z 207.065,A -85,B 0,C 180,E1 -614.409,E2 -614.409} C_VEL
LIN {X 0,Y 601.417,Z 207.073,A -85,B 0,C 180,E1 -617.172,E2 -617.172} C_VEL
LIN {X 0,Y 601.437,Z 207.063,A -85,B 0,C 180,E1 -619.905,E2 -619.905} C_VEL
LIN {X 0,Y 601.437,Z 207.064,A -85,B 0,C 180,E1 -622.615,E2 -622.615} C_VEL
LIN {X 0,Y 601.418,Z 207.071,A -85,B 0,C 180,E1 -625.308,E2 -625.308} C_VEL
LIN {X 0,Y 601.437,Z 207.062,A -85,B 0,C 180,E1 -627.991,E2 -627.991} C_VEL
LIN {X 0,Y 601.446,Z 207.066,A -85,B 0,C 180,E1 -630.67,E2 -630.67} C_VEL
LIN {X 0,Y 601.426,Z 207.067,A -85,B 0,C 180,E1 -633.35,E2 -633.35} C_VEL
LIN {X 0,Y 601.441,Z 207.061,A -85,B 0,C 180,E1 -636.037,E2 -636.037} C_VEL
LIN {X 0,Y 601.432,Z 207.072,A -85,B 0,C 180,E1 -638.738,E2 -638.738} C_VEL
LIN {X 0,Y 601.431,Z 207.064,A -85,B 0,C 180,E1 -641.458,E2 -641.458} C_VEL
LIN {X 0,Y 601.416,Z 207.067,A -85,B 0,C 180,E1 -644.205,E2 -644.205} C_VEL
LIN {X 0,Y 601.431,Z 207.067,A -85,B 0,C 180,E1 -646.986,E2 -646.986} C_VEL
LIN {X 0,Y 601.402,Z 207.066,A -85,B 0,C 180,E1 -649.809,E2 -649.809} C_VEL
LIN {X 0,Y 601.412,Z 207.074,A -85,B 0,C 180,E1 -652.606,E2 -652.606} C_VEL
LIN {X 0,Y 601.4,Z 207.07,A -85,B 0,C 180,E1 -654.879,E2 -654.879} C_VEL
LIN {X 0,Y 601.42,Z 207.066,A -85,B 0,C 180,E1 -657.867,E2 -657.867} C_VEL
LIN {X 0,Y 601.424,Z 207.069,A -85,B 0,C 180,E1 -660.164,E2 -660.164} C_VEL
LIN {X 0,Y 601.425,Z 207.067,A -85,B 0,C 180,E1 -662.717,E2 -662.717} C_VEL
LIN {X 0,Y 601.392,Z 207.067,A -85,B 0,C 180,E1 -665.112,E2 -665.112} C_VEL
LIN {X 0,Y 601.433,Z 207.062,A -85,B 0,C 180,E1 -667.419,E2 -667.419} C_VEL
LIN {X 0,Y 601.409,Z 207.072,A -85,B 0,C 180,E1 -669.995,E2 -669.995} C_VEL
LIN {X 0,Y 601.41,Z 207.066,A -85,B 0,C 180,E1 -672.67,E2 -672.67} C_VEL
LIN {X 0,Y 601.422,Z 207.065,A -85,B 0,C 180,E1 -675.482,E2 -675.482} C_VEL
LIN {X 0,Y 601.423,Z 207.067,A -85,B 0,C 180,E1 -678.407,E2 -678.407} C_VEL
LIN {X 0,Y 601.436,Z 207.062,A -85,B 0,C 180,E1 -680.876,E2 -680.876} C_VEL
LIN {X 0,Y 601.44,Z 207.068,A -85,B 0,C 180,E1 -683.734,E2 -683.734} C_VEL
LIN {X 0,Y 601.426,Z 207.063,A -85,B 0,C 180,E1 -686.687,E2 -686.687} C_VEL
LIN {X 0,Y 601.428,Z 207.063,A -85,B 0,C 180,E1 -689.059,E2 -689.059} C_VEL
LIN {X 0,Y 601.424,Z 207.067,A -85,B 0,C 180,E1 -691.373,E2 -691.373} C_VEL
LIN {X 0,Y 601.398,Z 207.074,A -85,B 0,C 180,E1 -693.637,E2 -693.637} C_VEL
LIN {X 0,Y 601.416,Z 207.064,A -85,B 0,C 180,E1 -696.59,E2 -696.59} C_VEL
LIN {X 0,Y 601.429,Z 207.07,A -85,B 0,C 180,E1 -699.479,E2 -699.479} C_VEL
LIN {X 0,Y 601.392,Z 207.067,A -85,B 0,C 180,E1 -702.312,E2 -702.312} C_VEL
LIN {X 0,Y 601.408,Z 207.065,A -85,B 0,C 180,E1 -704.409,E2 -704.409} C_VEL
LIN {X 0,Y 601.417,Z 207.07,A -85,B 0,C 180,E1 -707.172,E2 -707.172} C_VEL
LIN {X 0,Y 601.439,Z 207.063,A -85,B 0,C 180,E1 -709.905,E2 -709.905} C_VEL
LIN {X 0,Y 601.405,Z 207.066,A -85,B 0,C 180,E1 -712.615,E2 -712.615} C_VEL
LIN {X 0,Y 601.425,Z 207.073,A -85,B 0,C 180,E1 -715.308,E2 -715.308} C_VEL
LIN {X 0,Y 601.438,Z 207.061,A -85,B 0,C 180,E1 -717.991,E2 -717.991} C_VEL
LIN {X 0,Y 601.438,Z 207.063,A -85,B 0,C 180,E1 -720.67,E2 -720.67} C_VEL
LIN {X 0,Y 601.435,Z 207.068,A -85,B 0,C 180,E1 -723.35,E2 -723.35} C_VEL
LIN {X 0,Y 601.435,Z 207.062,A -85,B 0,C 180,E1 -726.037,E2 -726.037} C_VEL
LIN {X 0,Y 601.407,Z 207.07,A -85,B 0,C 180,E1 -728.738,E2 -728.738} C_VEL
LIN {X 0,Y 601.435,Z 207.064,A -85,B 0,C 180,E1 -731.458,E2 -731.458} C_VEL
LIN {X 0,Y 601.419,Z 207.065,A -85,B 0,C 180,E1 -734.206,E2 -734.206} C_VEL
LIN {X 0,Y 601.42,Z 207.071,A -85,B 0,C 180,E1 -736.987,E2 -736.987} C_VEL
LIN {X 0,Y 601.4,Z 207.065,A -85,B 0,C 180,E1 -739.81,E2 -739.81} C_VEL
LIN {X 0,Y 601.413,Z 207.074,A -85,B 0,C 180,E1 -742.683,E2 -742.683} C_VEL
LIN {X 0,Y 601.399,Z 207.073,A -85,B 0,C 180,E1 -744.879,E2 -744.879} C_VEL
LIN {X 0,Y 601.415,Z 207.064,A -85,B 0,C 180,E1 -747.363,E2 -747.363} C_VEL
LIN {X 0,Y 601.413,Z 207.065,A -85,B 0,C 180,E1 -749.394,E2 -749.394} C_VEL
LIN {X 0,Y 601.398,Z 207.066,A -85,B 0,C 180,E1 -751.727,E2 -751.727} C_VEL
LIN {X 0,Y 601.419,Z 207.067,A -85,B 0,C 180,E1 -754.119,E2 -754.119} C_VEL
LIN {X 0,Y 601.437,Z 207.062,A -85,B 0,C 180,E1 -757.383,E2 -757.383} C_VEL
LIN {X 0,Y 601.401,Z 207.069,A -85,B 0,C 180,E1 -759.996,E2 -759.996} C_VEL
LIN {X 0,Y 601.417,Z 207.069,A -85,B 0,C 180,E1 -762.67,E2 -762.67} C_VEL
LIN {X 0,Y 601.399,Z 207.066,A -85,B 0,C 180,E1 -765.48,E2 -765.48} C_VEL
LIN {X 0,Y 601.424,Z 207.07,A -85,B 0,C 180,E1 -768.407,E2 -768.407} C_VEL
LIN {X 0,Y 601.432,Z 207.063,A -85,B 0,C 180,E1 -770.875,E2 -770.875} C_VEL
LIN {X 0,Y 601.399,Z 207.067,A -85,B 0,C 180,E1 -773.417,E2 -773.417} C_VEL
LIN {X 0,Y 601.432,Z 207.073,A -85,B 0,C 180,E1 -776.065,E2 -776.065} C_VEL
LIN {X 0,Y 601.411,Z 207.065,A -85,B 0,C 180,E1 -779.058,E2 -779.058} C_VEL
LIN {X 0,Y 601.414,Z 207.067,A -85,B 0,C 180,E1 -781.372,E2 -781.372} C_VEL
LIN {X 0,Y 601.411,Z 207.073,A -85,B 0,C 180,E1 -784.134,E2 -784.134} C_VEL
LIN {X 0,Y 601.461,Z 207.238,A -85,B 0,C 180,E1 -785.703,E2 -785.703} C_VEL
LIN {X 0,Y 601.562,Z 216.544,A -85,B 0,C 180,E1 -787.362,E2 -787.362} C_VEL
LIN {X 0,Y 601.529,Z 231.845,A -85,B 0,C 180,E1 -790.017,E2 -790.017} C_VEL
LIN {X 0,Y 601.468,Z 248.402,A -85,B 0,C 180,E1 -792.84,E2 -792.84} C_VEL
LIN {X 0,Y 601.456,Z 263.924,A -85,B 0,C 180,E1 -795.45,E2 -795.45} C_VEL
LIN {X 0,Y 601.451,Z 272.24,A -85,B 0,C 180,E1 -796.808,E2 -796.808} C_VEL
LIN {X 0,Y 601.633,Z 274.724,A -85,B 0,C 180,E1 -796.876,E2 -796.876} C_VEL
LIN {X 0,Y 601.617,Z 378.889,A -85,B 0,C 180,E1 -798.14,E2 -798.14} C_VEL
LIN {X 0,Y 601.591,Z 392.237,A -85,B 0,C 180,E1 -798.438,E2 -798.438} C_VEL
LIN {X 0,Y 601.547,Z 404.665,A -85,B 0,C 180,E1 -798.854,E2 -798.854} C_VEL
LIN {X 0,Y 601.52,Z 416.603,A -85,B 0,C 180,E1 -799.396,E2 -799.396} C_VEL
LIN {X 0,Y 601.484,Z 428.201,A -85,B 0,C 180,E1 -800.076,E2 -800.076} C_VEL
LIN {X 0,Y 601.438,Z 439.645,A -85,B 0,C 180,E1 -800.924,E2 -800.924} C_VEL
LIN {X 0,Y 601.411,Z 448.775,A -85,B 0,C 180,E1 -801.77,E2 -801.77} C_VEL
LIN {X 0,Y 601.388,Z 457.681,A -85,B 0,C 180,E1 -802.783,E2 -802.783} C_VEL
LIN {X 0,Y 601.375,Z 464.773,A -85,B 0,C 180,E1 -803.782,E2 -803.782} C_VEL
LIN {X 0,Y 601.345,Z 471.364,A -85,B 0,C 180,E1 -804.971,E2 -804.971} C_VEL
LIN {X 0,Y 601.347,Z 475.671,A -85,B 0,C 180,E1 -805.979,E2 -805.979} C_VEL
LIN {X 0,Y 601.344,Z 477.959,A -85,B 0,C 180,E1 -806.65,E2 -806.65} C_VEL
LIN {X 0,Y 601.325,Z 479.804,A -85,B 0,C 180,E1 -807.32,E2 -807.32} C_VEL
LIN {X 0,Y 601.343,Z 481.198,A -85,B 0,C 180,E1 -807.991,E2 -807.991} C_VEL
LIN {X 0,Y 601.339,Z 482.783,A -85,B 0,C 180,E1 -809.33,E2 -809.33} C_VEL
LIN {X 0,Y 601.335,Z 482.989,A -85,B 0,C 180,E1 -810,E2 -810} C_VEL
LIN {X 0,Y 601.347,Z 482.186,A -85,B 0,C 180,E1 -811.339,E2 -811.339} C_VEL
LIN {X 0,Y 601.343,Z 481.198,A -85,B 0,C 180,E1 -812.009,E2 -812.009} C_VEL
LIN {X 0,Y 601.325,Z 479.804,A -85,B 0,C 180,E1 -812.68,E2 -812.68} C_VEL
LIN {X 0,Y 601.368,Z 476.893,A -85,B 0,C 180,E1 -813.685,E2 -813.685} C_VEL
LIN {X 0,Y 601.336,Z 472.948,A -85,B 0,C 180,E1 -814.693,E2 -814.693} C_VEL
LIN {X 0,Y 601.374,Z 467.855,A -85,B 0,C 180,E1 -815.701,E2 -815.701} C_VEL
LIN {X 0,Y 601.382,Z 461.469,A -85,B 0,C 180,E1 -816.711,E2 -816.711} C_VEL
LIN {X 0,Y 601.396,Z 453.483,A -85,B 0,C 180,E1 -817.723,E2 -817.723} C_VEL
LIN {X 0,Y 601.423,Z 445.342,A -85,B 0,C 180,E1 -818.568,E2 -818.568} C_VEL
LIN {X 0,Y 601.454,Z 435.381,A -85,B 0,C 180,E1 -819.415,E2 -819.415} C_VEL
LIN {X 0,Y 601.48,Z 425.567,A -85,B 0,C 180,E1 -820.094,E2 -820.094} C_VEL
LIN {X 0,Y 601.53,Z 414.93,A -85,B 0,C 180,E1 -820.689,E2 -820.689} C_VEL
LIN {X 0,Y 601.572,Z 401.568,A -85,B 0,C 180,E1 -821.263,E2 -821.263} C_VEL
LIN {X 0,Y 601.593,Z 389.032,A -85,B 0,C 180,E1 -821.647,E2 -821.647} C_VEL
LIN {X 0,Y 601.634,Z 376.111,A -85,B 0,C 180,E1 -821.903,E2 -821.903} C_VEL
LIN {X 0,Y 601.526,Z 273.222,A -85,B 0,C 180,E1 -823.148,E2 -823.148} C_VEL
LIN {X 0,Y 601.415,Z 272.027,A -85,B 0,C 180,E1 -823.215,E2 -823.215} C_VEL
LIN {X 0,Y 601.487,Z 255.645,A -85,B 0,C 180,E1 -825.937,E2 -825.937} C_VEL
LIN {X 0,Y 601.525,Z 238.464,A -85,B 0,C 180,E1 -828.848,E2 -828.848} C_VEL
LIN {X 0,Y 601.557,Z 222.532,A -85,B 0,C 180,E1 -831.593,E2 -831.593} C_VEL
LIN {X 0,Y 601.601,Z 208.045,A -85,B 0,C 180,E1 -834.134,E2 -834.134} C_VEL
LIN {X 0,Y 601.421,Z 207.11,A -85,B 0,C 180,E1 -834.383,E2 -834.383} C_VEL
LIN {X 0,Y 601.423,Z 207.064,A -85,B 0,C 180,E1 -837.112,E2 -837.112} C_VEL
LIN {X 0,Y 601.431,Z 207.071,A -85,B 0,C 180,E1 -840.148,E2 -840.148} C_VEL
LIN {X 0,Y 601.41,Z 207.065,A -85,B 0,C 180,E1 -842.713,E2 -842.713} C_VEL
LIN {X 0,Y 601.389,Z 207.068,A -85,B 0,C 180,E1 -845.111,E2 -845.111} C_VEL
LIN {X 0,Y 601.437,Z 207.065,A -85,B 0,C 180,E1 -847.419,E2 -847.419} C_VEL
LIN {X 0,Y 601.414,Z 207.071,A -85,B 0,C 180,E1 -849.995,E2 -849.995} C_VEL
LIN {X 0,Y 601.407,Z 207.065,A -85,B 0,C 180,E1 -852.67,E2 -852.67} C_VEL
LIN {X 0,Y 601.428,Z 207.069,A -85,B 0,C 180,E1 -855.482,E2 -855.482} C_VEL
LIN {X 0,Y 601.418,Z 207.064,A -85,B 0,C 180,E1 -858.407,E2 -858.407} C_VEL
LIN {X 0,Y 601.414,Z 207.065,A -85,B 0,C 180,E1 -860.873,E2 -860.873} C_VEL
LIN {X 0,Y 601.404,Z 207.074,A -85,B 0,C 180,E1 -863.417,E2 -863.417} C_VEL
LIN {X 0,Y 601.416,Z 207.065,A -85,B 0,C 180,E1 -866.066,E2 -866.066} C_VEL
LIN {X 0,Y 601.419,Z 207.064,A -85,B 0,C 180,E1 -868.545,E2 -868.545} C_VEL
LIN {X 0,Y 601.432,Z 207.072,A -85,B 0,C 180,E1 -871.373,E2 -871.373} C_VEL
LIN {X 0,Y 601.397,Z 207.071,A -85,B 0,C 180,E1 -873.636,E2 -873.636} C_VEL
LIN {X 0,Y 601.417,Z 207.065,A -85,B 0,C 180,E1 -876.589,E2 -876.589} C_VEL
LIN {X 0,Y 601.424,Z 207.068,A -85,B 0,C 180,E1 -879.478,E2 -879.478} C_VEL
LIN {X 0,Y 601.391,Z 207.066,A -85,B 0,C 180,E1 -882.311,E2 -882.311} C_VEL
LIN {X 0,Y 601.411,Z 207.065,A -85,B 0,C 180,E1 -884.408,E2 -884.408} C_VEL
LIN {X 0,Y 601.412,Z 207.073,A -85,B 0,C 180,E1 -887.171,E2 -887.171} C_VEL
LIN {X 0,Y 601.433,Z 207.061,A -85,B 0,C 180,E1 -889.905,E2 -889.905} C_VEL
LIN {X 0,Y 601.443,Z 207.065,A -85,B 0,C 180,E1 -892.615,E2 -892.615} C_VEL
LIN {X 0,Y 601.41,Z 207.069,A -85,B 0,C 180,E1 -895.308,E2 -895.308} C_VEL
LIN {X 0,Y 601.436,Z 207.061,A -85,B 0,C 180,E1 -897.991,E2 -897.991} C_VEL
LIN {X 0,Y 601.455,Z 207.066,A -85,B 0,C 180,E1 -900.669,E2 -900.669} C_VEL
LIN {X 0,Y 601.417,Z 207.065,A -85,B 0,C 180,E1 -903.349,E2 -903.349} C_VEL
LIN {X 0,Y 601.442,Z 207.062,A -85,B 0,C 180,E1 -906.036,E2 -906.036} C_VEL
LIN {X 0,Y 601.437,Z 207.069,A -85,B 0,C 180,E1 -908.737,E2 -908.737} C_VEL
LIN {X 0,Y 601.411,Z 207.064,A -85,B 0,C 180,E1 -911.458,E2 -911.458} C_VEL
LIN {X 0,Y 601.408,Z 207.068,A -85,B 0,C 180,E1 -912.376,E2 -912.376} C_VEL
LIN {X 0,Y 600.742,Z 207.153,A -85,B 0,C 180,E1 -912.936,E2 -912.936} C_VEL
LIN {X 0,Y 597.891,Z 207.507,A -85,B 0,C 180,E1 -913.844,E2 -913.844} C_VEL
LIN {X 0,Y 595.481,Z 207.813,A -85,B 0,C 180,E1 -914.574,E2 -914.574} C_VEL
LIN {X 0,Y 594.444,Z 207.935,A -85,B 0,C 180,E1 -915.137,E2 -915.137} C_VEL
LIN {X 0,Y 594.358,Z 207.944,A -85,B 0,C 180,E1 -915.328,E2 -915.328} C_VEL
LIN {X 0,Y 594.386,Z 207.94,A -85,B 0,C 180,E1 -917.193,E2 -917.193} C_VEL
LIN {X 0,Y 594.373,Z 207.944,A -85,B 0,C 180,E1 -920.053,E2 -920.053} C_VEL
LIN {X 0,Y 594.355,Z 207.945,A -85,B 0,C 180,E1 -922.967,E2 -922.967} C_VEL
LIN {X 0,Y 594.374,Z 207.941,A -85,B 0,C 180,E1 -925.193,E2 -925.193} C_VEL
LIN {X 0,Y 594.383,Z 207.939,A -85,B 0,C 180,E1 -927.526,E2 -927.526} C_VEL
LIN {X 0,Y 594.385,Z 207.948,A -85,B 0,C 180,E1 -930.328,E2 -930.328} C_VEL
LIN {X 0,Y 594.376,Z 207.941,A -85,B 0,C 180,E1 -932.95,E2 -932.95} C_VEL
LIN {X 0,Y 594.351,Z 207.944,A -85,B 0,C 180,E1 -935.408,E2 -935.408} C_VEL
LIN {X 0,Y 594.386,Z 207.949,A -85,B 0,C 180,E1 -937.94,E2 -937.94} C_VEL
LIN {X 0,Y 594.377,Z 207.94,A -85,B 0,C 180,E1 -940.822,E2 -940.822} C_VEL
LIN {X 0,Y 594.38,Z 207.95,A -85,B 0,C 180,E1 -943.841,E2 -943.841} C_VEL
LIN {X 0,Y 594.377,Z 207.939,A -85,B 0,C 180,E1 -946.702,E2 -946.702} C_VEL
LIN {X 0,Y 594.371,Z 207.944,A -85,B 0,C 180,E1 -949.433,E2 -949.433} C_VEL
LIN {X 0,Y 594.388,Z 207.941,A -85,B 0,C 180,E1 -952.391,E2 -952.391} C_VEL
LIN {X 0,Y 594.349,Z 207.943,A -85,B 0,C 180,E1 -954.676,E2 -954.676} C_VEL
LIN {X 0,Y 594.378,Z 207.942,A -85,B 0,C 180,E1 -957.088,E2 -957.088} C_VEL
LIN {X 0,Y 594.384,Z 207.948,A -85,B 0,C 180,E1 -959.671,E2 -959.671} C_VEL
LIN {X 0,Y 594.371,Z 207.942,A -85,B 0,C 180,E1 -962.539,E2 -962.539} C_VEL
LIN {X 0,Y 594.372,Z 207.943,A -85,B 0,C 180,E1 -964.807,E2 -964.807} C_VEL
LIN {X 0,Y 594.362,Z 207.95,A -85,B 0,C 180,E1 -967.264,E2 -967.264} C_VEL
LIN {X 0,Y 594.372,Z 207.944,A -85,B 0,C 180,E1 -969.946,E2 -969.946} C_VEL
LIN {X 0,Y 594.387,Z 207.942,A -85,B 0,C 180,E1 -972.807,E2 -972.807} C_VEL
LIN {X 0,Y 594.386,Z 207.943,A -85,B 0,C 180,E1 -975.826,E2 -975.826} C_VEL
LIN {X 0,Y 594.391,Z 207.94,A -85,B 0,C 180,E1 -978.404,E2 -978.404} C_VEL
LIN {X 0,Y 594.394,Z 207.949,A -85,B 0,C 180,E1 -981.158,E2 -981.158} C_VEL
LIN {X 0,Y 594.394,Z 207.94,A -85,B 0,C 180,E1 -983.891,E2 -983.891} C_VEL
LIN {X 0,Y 594.378,Z 207.945,A -85,B 0,C 180,E1 -986.611,E2 -986.611} C_VEL
LIN {X 0,Y 594.417,Z 207.942,A -85,B 0,C 180,E1 -989.323,E2 -989.323} C_VEL
LIN {X 0,Y 594.406,Z 207.938,A -85,B 0,C 180,E1 -992.033,E2 -992.033} C_VEL
LIN {X 0,Y 594.387,Z 207.948,A -85,B 0,C 180,E1 -994.748,E2 -994.748} C_VEL
LIN {X 0,Y 594.391,Z 207.941,A -85,B 0,C 180,E1 -997.473,E2 -997.473} C_VEL
LIN {X 0,Y 594.396,Z 207.941,A -85,B 0,C 180,E1 -1000.216,E2 -1000.216} C_VEL
LIN {X 0,Y 594.364,Z 207.949,A -85,B 0,C 180,E1 -1002.983,E2 -1002.983} C_VEL
LIN {X 0,Y 594.364,Z 207.943,A -85,B 0,C 180,E1 -1005.781,E2 -1005.781} C_VEL
LIN {X 0,Y 594.385,Z 207.951,A -85,B 0,C 180,E1 -1008.617,E2 -1008.617} C_VEL
LIN {X 0,Y 594.367,Z 207.943,A -85,B 0,C 180,E1 -1011.503,E2 -1011.503} C_VEL
LIN {X 0,Y 594.385,Z 207.95,A -85,B 0,C 180,E1 -1014.446,E2 -1014.446} C_VEL
LIN {X 0,Y 594.383,Z 207.947,A -85,B 0,C 180,E1 -1016.699,E2 -1016.699} C_VEL
LIN {X 0,Y 594.38,Z 207.941,A -85,B 0,C 180,E1 -1018.998,E2 -1018.998} C_VEL
LIN {X 0,Y 594.39,Z 207.94,A -85,B 0,C 180,E1 -1021.645,E2 -1021.645} C_VEL
LIN {X 0,Y 594.377,Z 207.945,A -85,B 0,C 180,E1 -1024.58,E2 -1024.58} C_VEL
LIN {X 0,Y 594.383,Z 207.941,A -85,B 0,C 180,E1 -1027.087,E2 -1027.087} C_VEL
LIN {X 0,Y 594.373,Z 207.945,A -85,B 0,C 180,E1 -1029.775,E2 -1029.775} C_VEL
LIN {X 0,Y 594.368,Z 207.947,A -85,B 0,C 180,E1 -1032.375,E2 -1032.375} C_VEL
LIN {X 0,Y 594.36,Z 207.943,A -85,B 0,C 180,E1 -1035.191,E2 -1035.191} C_VEL
LIN {X 0,Y 594.365,Z 207.946,A -85,B 0,C 180,E1 -1037.625,E2 -1037.625} C_VEL
LIN {X 0,Y 594.39,Z 207.944,A -85,B 0,C 180,E1 -1040.321,E2 -1040.321} C_VEL
LIN {X 0,Y 594.384,Z 207.94,A -85,B 0,C 180,E1 -1042.914,E2 -1042.914} C_VEL
LIN {X 0,Y 594.379,Z 207.95,A -85,B 0,C 180,E1 -1045.862,E2 -1045.862} C_VEL
LIN {X 0,Y 594.387,Z 207.94,A -85,B 0,C 180,E1 -1048.651,E2 -1048.651} C_VEL
LIN {X 0,Y 594.379,Z 207.941,A -85,B 0,C 180,E1 -1051.042,E2 -1051.042} C_VEL
LIN {X 0,Y 594.385,Z 207.946,A -85,B 0,C 180,E1 -1053.977,E2 -1053.977} C_VEL
LIN {X 0,Y 594.388,Z 207.941,A -85,B 0,C 180,E1 -1056.296,E2 -1056.296} C_VEL
LIN {X 0,Y 594.401,Z 207.942,A -85,B 0,C 180,E1 -1059.225,E2 -1059.225} C_VEL
LIN {X 0,Y 594.35,Z 207.946,A -85,B 0,C 180,E1 -1062.095,E2 -1062.095} C_VEL
LIN {X 0,Y 594.363,Z 207.943,A -85,B 0,C 180,E1 -1064.219,E2 -1064.219} C_VEL
LIN {X 0,Y 594.377,Z 207.941,A -85,B 0,C 180,E1 -1066.321,E2 -1066.321} C_VEL
LIN {X 0,Y 594.374,Z 207.945,A -85,B 0,C 180,E1 -1069.095,E2 -1069.095} C_VEL
LIN {X 0,Y 594.418,Z 207.938,A -85,B 0,C 180,E1 -1071.844,E2 -1071.844} C_VEL
LIN {X 0,Y 594.387,Z 207.94,A -85,B 0,C 180,E1 -1074.573,E2 -1074.573} C_VEL
LIN {X 0,Y 594.408,Z 207.946,A -85,B 0,C 180,E1 -1077.29,E2 -1077.29} C_VEL
LIN {X 0,Y 594.414,Z 207.935,A -85,B 0,C 180,E1 -1080,E2 -1080} C_VEL
LIN {X 0,Y 594.395,Z 207.942,A -85,B 0,C 180,E1 -1082.711,E2 -1082.711} C_VEL
LIN {X 0,Y 594.4,Z 207.943,A -85,B 0,C 180,E1 -1085.428,E2 -1085.428} C_VEL
LIN {X 0,Y 594.382,Z 207.939,A -85,B 0,C 180,E1 -1088.158,E2 -1088.158} C_VEL
LIN {X 0,Y 594.387,Z 207.948,A -85,B 0,C 180,E1 -1091.073,E2 -1091.073} C_VEL
LIN {X 0,Y 594.379,Z 207.941,A -85,B 0,C 180,E1 -1093.679,E2 -1093.679} C_VEL
LIN {X 0,Y 594.385,Z 207.947,A -85,B 0,C 180,E1 -1096.717,E2 -1096.717} C_VEL
LIN {X 0,Y 594.365,Z 207.944,A -85,B 0,C 180,E1 -1099.335,E2 -1099.335} C_VEL
LIN {X 0,Y 594.364,Z 207.943,A -85,B 0,C 180,E1 -1101.504,E2 -1101.504} C_VEL
LIN {X 0,Y 594.388,Z 207.945,A -85,B 0,C 180,E1 -1104.446,E2 -1104.446} C_VEL
LIN {X 0,Y 594.382,Z 207.949,A -85,B 0,C 180,E1 -1106.7,E2 -1106.7} C_VEL
LIN {X 0,Y 594.381,Z 207.944,A -85,B 0,C 180,E1 -1108.999,E2 -1108.999} C_VEL
LIN {X 0,Y 594.376,Z 207.941,A -85,B 0,C 180,E1 -1111.643,E2 -1111.643} C_VEL
LIN {X 0,Y 594.378,Z 207.95,A -85,B 0,C 180,E1 -1114.58,E2 -1114.58} C_VEL
LIN {X 0,Y 594.389,Z 207.94,A -85,B 0,C 180,E1 -1117.609,E2 -1117.609} C_VEL
LIN {X 0,Y 594.367,Z 207.949,A -85,B 0,C 180,E1 -1120.567,E2 -1120.567} C_VEL
LIN {X 0,Y 594.368,Z 207.942,A -85,B 0,C 180,E1 -1123.3,E2 -1123.3} C_VEL
LIN {X 0,Y 594.362,Z 207.951,A -85,B 0,C 180,E1 -1126.162,E2 -1126.162} C_VEL
LIN {X 0,Y 594.381,Z 207.944,A -85,B 0,C 180,E1 -1128.536,E2 -1128.536} C_VEL
LIN {X 0,Y 594.378,Z 207.941,A -85,B 0,C 180,E1 -1131.297,E2 -1131.297} C_VEL
LIN {X 0,Y 594.351,Z 207.948,A -85,B 0,C 180,E1 -1133.756,E2 -1133.756} C_VEL
LIN {X 0,Y 594.378,Z 207.948,A -85,B 0,C 180,E1 -1136.239,E2 -1136.239} C_VEL
LIN {X 0,Y 594.37,Z 207.944,A -85,B 0,C 180,E1 -1138.65,E2 -1138.65} C_VEL
LIN {X 0,Y 594.378,Z 207.942,A -85,B 0,C 180,E1 -1141.044,E2 -1141.044} C_VEL
LIN {X 0,Y 594.369,Z 207.945,A -85,B 0,C 180,E1 -1143.3,E2 -1143.3} C_VEL
LIN {X 0,Y 594.401,Z 208.166,A -85,B 0,C 180,E1 -1145.564,E2 -1145.564} C_VEL
LIN {X 0,Y 594.665,Z 212.184,A -85,B 0,C 180,E1 -1146.308,E2 -1146.308} C_VEL
LIN {X 0,Y 594.542,Z 228.741,A -85,B 0,C 180,E1 -1149.23,E2 -1149.23} C_VEL
LIN {X 0,Y 594.48,Z 244.263,A -85,B 0,C 180,E1 -1151.921,E2 -1151.921} C_VEL
LIN {X 0,Y 594.398,Z 260.819,A -85,B 0,C 180,E1 -1154.747,E2 -1154.747} C_VEL
LIN {X 0,Y 594.409,Z 272.235,A -85,B 0,C 180,E1 -1156.648,E2 -1156.648} C_VEL
LIN {X 0,Y 594.725,Z 274.724,A -85,B 0,C 180,E1 -1156.721,E2 -1156.721} C_VEL
LIN {X 0,Y 594.669,Z 378.828,A -85,B 0,C 180,E1 -1157.999,E2 -1157.999} C_VEL
LIN {X 0,Y 594.626,Z 391.488,A -85,B 0,C 180,E1 -1158.279,E2 -1158.279} C_VEL
LIN {X 0,Y 594.576,Z 405.331,A -85,B 0,C 180,E1 -1158.748,E2 -1158.748} C_VEL
LIN {X 0,Y 594.537,Z 416.583,A -85,B 0,C 180,E1 -1159.27,E2 -1159.27} C_VEL
LIN {X 0,Y 594.454,Z 426.898,A -85,B 0,C 180,E1 -1159.871,E2 -1159.871} C_VEL
LIN {X 0,Y 594.405,Z 437.544,A -85,B 0,C 180,E1 -1160.644,E2 -1160.644} C_VEL
LIN {X 0,Y 594.383,Z 447.12,A -85,B 0,C 180,E1 -1161.501,E2 -1161.501} C_VEL
LIN {X 0,Y 594.347,Z 454.946,A -85,B 0,C 180,E1 -1162.355,E2 -1162.355} C_VEL
LIN {X 0,Y 594.303,Z 462.692,A -85,B 0,C 180,E1 -1163.391,E2 -1163.391} C_VEL
LIN {X 0,Y 594.289,Z 469.681,A -85,B 0,C 180,E1 -1164.571,E2 -1164.571} C_VEL
LIN {X 0,Y 594.27,Z 474.376,A -85,B 0,C 180,E1 -1165.591,E2 -1165.591} C_VEL
LIN {X 0,Y 594.267,Z 477.962,A -85,B 0,C 180,E1 -1166.61,E2 -1166.61} C_VEL
LIN {X 0,Y 594.225,Z 479.798,A -85,B 0,C 180,E1 -1167.288,E2 -1167.288} C_VEL
LIN {X 0,Y 594.242,Z 481.191,A -85,B 0,C 180,E1 -1167.967,E2 -1167.967} C_VEL
LIN {X 0,Y 594.247,Z 482.188,A -85,B 0,C 180,E1 -1168.645,E2 -1168.645} C_VEL
LIN {X 0,Y 594.239,Z 482.782,A -85,B 0,C 180,E1 -1169.322,E2 -1169.322} C_VEL
LIN {X 0,Y 594.236,Z 482.98,A -85,B 0,C 180,E1 -1170,E2 -1170} C_VEL
LIN {X 0,Y 594.239,Z 482.782,A -85,B 0,C 180,E1 -1170.678,E2 -1170.678} C_VEL
LIN {X 0,Y 594.247,Z 482.188,A -85,B 0,C 180,E1 -1171.355,E2 -1171.355} C_VEL
LIN {X 0,Y 594.242,Z 481.191,A -85,B 0,C 180,E1 -1172.033,E2 -1172.033} C_VEL
LIN {X 0,Y 594.225,Z 479.798,A -85,B 0,C 180,E1 -1172.712,E2 -1172.712} C_VEL
LIN {X 0,Y 594.289,Z 476.888,A -85,B 0,C 180,E1 -1173.729,E2 -1173.729} C_VEL
LIN {X 0,Y 594.241,Z 472.939,A -85,B 0,C 180,E1 -1174.749,E2 -1174.749} C_VEL
LIN {X 0,Y 594.3,Z 467.844,A -85,B 0,C 180,E1 -1175.769,E2 -1175.769} C_VEL
LIN {X 0,Y 594.316,Z 461.461,A -85,B 0,C 180,E1 -1176.791,E2 -1176.791} C_VEL
LIN {X 0,Y 594.346,Z 453.487,A -85,B 0,C 180,E1 -1177.816,E2 -1177.816} C_VEL
LIN {X 0,Y 594.378,Z 445.346,A -85,B 0,C 180,E1 -1178.671,E2 -1178.671} C_VEL
LIN {X 0,Y 594.417,Z 435.367,A -85,B 0,C 180,E1 -1179.528,E2 -1179.528} C_VEL
LIN {X 0,Y 594.469,Z 425.549,A -85,B 0,C 180,E1 -1180.215,E2 -1180.215} C_VEL
LIN {X 0,Y 594.55,Z 414.935,A -85,B 0,C 180,E1 -1180.816,E2 -1180.816} C_VEL
LIN {X 0,Y 594.598,Z 402.052,A -85,B 0,C 180,E1 -1181.379,E2 -1181.379} C_VEL
LIN {X 0,Y 594.654,Z 389.869,A -85,B 0,C 180,E1 -1181.763,E2 -1181.763} C_VEL
LIN {X 0,Y 594.675,Z 377.497,A -85,B 0,C 180,E1 -1182.022,E2 -1182.022} C_VEL
LIN {X 0,Y 594.573,Z 273.647,A -85,B 0,C 180,E1 -1183.296,E2 -1183.296} C_VEL
LIN {X 0,Y 594.398,Z 272.025,A -85,B 0,C 180,E1 -1183.374,E2 -1183.374} C_VEL
LIN {X 0,Y 594.449,Z 255.645,A -85,B 0,C 180,E1 -1186.131,E2 -1186.131} C_VEL
LIN {X 0,Y 594.531,Z 239.093,A -85,B 0,C 180,E1 -1188.97,E2 -1188.97} C_VEL
LIN {X 0,Y 594.585,Z 223.567,A -85,B 0,C 180,E1 -1191.677,E2 -1191.677} C_VEL
LIN {X 0,Y 594.67,Z 210.142,A -85,B 0,C 180,E1 -1194.057,E2 -1194.057} C_VEL
LIN {X 0,Y 594.386,Z 208.011,A -85,B 0,C 180,E1 -1194.493,E2 -1194.493} C_VEL
LIN {X 0,Y 594.378,Z 207.944,A -85,B 0,C 180,E1 -1197.461,E2 -1197.461} C_VEL
LIN {X 0,Y 594.387,Z 207.945,A -85,B 0,C 180,E1 -1200.328,E2 -1200.328} C_VEL
LIN {X 0,Y 594.377,Z 207.941,A -85,B 0,C 180,E1 -1202.95,E2 -1202.95} C_VEL
LIN {X 0,Y 594.35,Z 207.947,A -85,B 0,C 180,E1 -1205.409,E2 -1205.409} C_VEL
LIN {X 0,Y 594.382,Z 207.949,A -85,B 0,C 180,E1 -1207.941,E2 -1207.941} C_VEL
LIN {X 0,Y 594.374,Z 207.94,A -85,B 0,C 180,E1 -1210.821,E2 -1210.821} C_VEL
LIN {X 0,Y 594.367,Z 207.946,A -85,B 0,C 180,E1 -1213.299,E2 -1213.299} C_VEL
LIN {X 0,Y 594.368,Z 207.945,A -85,B 0,C 180,E1 -1216.16,E2 -1216.16} C_VEL
LIN {X 0,Y 594.377,Z 207.941,A -85,B 0,C 180,E1 -1218.535,E2 -1218.535} C_VEL
LIN {X 0,Y 594.382,Z 207.945,A -85,B 0,C 180,E1 -1221.296,E2 -1221.296} C_VEL
LIN {X 0,Y 594.35,Z 207.95,A -85,B 0,C 180,E1 -1223.755,E2 -1223.755} C_VEL
LIN {X 0,Y 594.365,Z 207.942,A -85,B 0,C 180,E1 -1226.238,E2 -1226.238} C_VEL
LIN {X 0,Y 594.369,Z 207.942,A -85,B 0,C 180,E1 -1228.649,E2 -1228.649} C_VEL
LIN {X 0,Y 594.384,Z 207.945,A -85,B 0,C 180,E1 -1231.042,E2 -1231.042} C_VEL
LIN {X 0,Y 594.38,Z 207.941,A -85,B 0,C 180,E1 -1233.978,E2 -1233.978} C_VEL
LIN {X 0,Y 594.383,Z 207.94,A -85,B 0,C 180,E1 -1236.295,E2 -1236.295} C_VEL
LIN {X 0,Y 594.402,Z 207.947,A -85,B 0,C 180,E1 -1239.224,E2 -1239.224} C_VEL
LIN {X 0,Y 594.344,Z 207.944,A -85,B 0,C 180,E1 -1242.094,E2 -1242.094} C_VEL
LIN {X 0,Y 594.362,Z 207.942,A -85,B 0,C 180,E1 -1244.219,E2 -1244.219} C_VEL
LIN {X 0,Y 594.379,Z 207.941,A -85,B 0,C 180,E1 -1246.321,E2 -1246.321} C_VEL
LIN {X 0,Y 594.371,Z 207.949,A -85,B 0,C 180,E1 -1249.094,E2 -1249.094} C_VEL
LIN {X 0,Y 594.382,Z 207.939,A -85,B 0,C 180,E1 -1251.842,E2 -1251.842} C_VEL
LIN {X 0,Y 594.4,Z 207.943,A -85,B 0,C 180,E1 -1254.572,E2 -1254.572} C_VEL
LIN {X 0,Y 594.395,Z 207.942,A -85,B 0,C 180,E1 -1257.289,E2 -1257.289} C_VEL
LIN {X 0,Y 594.414,Z 207.935,A -85,B 0,C 180,E1 -1260,E2 -1260} C_VEL
LIN {X 0,Y 594.408,Z 207.946,A -85,B 0,C 180,E1 -1262.71,E2 -1262.71} C_VEL
LIN {X 0,Y 594.388,Z 207.94,A -85,B 0,C 180,E1 -1265.427,E2 -1265.427} C_VEL
LIN {X 0,Y 594.418,Z 207.938,A -85,B 0,C 180,E1 -1268.156,E2 -1268.156} C_VEL
LIN {X 0,Y 594.388,Z 207.941,A -85,B 0,C 180,E1 -1271.074,E2 -1271.074} C_VEL
LIN {X 0,Y 594.377,Z 207.941,A -85,B 0,C 180,E1 -1273.679,E2 -1273.679} C_VEL
LIN {X 0,Y 594.358,Z 207.944,A -85,B 0,C 180,E1 -1275.328,E2 -1275.328} C_VEL
LIN {X 0,Y 593.683,Z 208.03,A -85,B 0,C 180,E1 -1275.894,E2 -1275.894} C_VEL
LIN {X 0,Y 590.818,Z 208.388,A -85,B 0,C 180,E1 -1276.812,E2 -1276.812} C_VEL
LIN {X 0,Y 588.408,Z 208.69,A -85,B 0,C 180,E1 -1277.551,E2 -1277.551} C_VEL
LIN {X 0,Y 587.385,Z 208.816,A -85,B 0,C 180,E1 -1278.121,E2 -1278.121} C_VEL
LIN {X 0,Y 587.308,Z 208.824,A -85,B 0,C 180,E1 -1278.314,E2 -1278.314} C_VEL
LIN {X 0,Y 587.328,Z 208.82,A -85,B 0,C 180,E1 -1281.037,E2 -1281.037} C_VEL
LIN {X 0,Y 587.313,Z 208.821,A -85,B 0,C 180,E1 -1283.259,E2 -1283.259} C_VEL
LIN {X 0,Y 587.333,Z 208.818,A -85,B 0,C 180,E1 -1285.516,E2 -1285.516} C_VEL
LIN {X 0,Y 587.344,Z 208.818,A -85,B 0,C 180,E1 -1287.817,E2 -1287.817} C_VEL
LIN {X 0,Y 587.34,Z 208.823,A -85,B 0,C 180,E1 -1290.511,E2 -1290.511} C_VEL
LIN {X 0,Y 587.337,Z 208.817,A -85,B 0,C 180,E1 -1293.112,E2 -1293.112} C_VEL
LIN {X 0,Y 587.315,Z 208.827,A -85,B 0,C 180,E1 -1295.898,E2 -1295.898} C_VEL
LIN {X 0,Y 587.331,Z 208.822,A -85,B 0,C 180,E1 -1298.479,E2 -1298.479} C_VEL
LIN {X 0,Y 587.335,Z 208.818,A -85,B 0,C 180,E1 -1301.156,E2 -1301.156} C_VEL
LIN {X 0,Y 587.331,Z 208.825,A -85,B 0,C 180,E1 -1304.114,E2 -1304.114} C_VEL
LIN {X 0,Y 587.319,Z 208.818,A -85,B 0,C 180,E1 -1306.994,E2 -1306.994} C_VEL
LIN {X 0,Y 587.317,Z 208.827,A -85,B 0,C 180,E1 -1309.746,E2 -1309.746} C_VEL
LIN {X 0,Y 587.343,Z 208.819,A -85,B 0,C 180,E1 -1312.392,E2 -1312.392} C_VEL
LIN {X 0,Y 587.322,Z 208.819,A -85,B 0,C 180,E1 -1314.944,E2 -1314.944} C_VEL
LIN {X 0,Y 587.339,Z 208.823,A -85,B 0,C 180,E1 -1317.421,E2 -1317.421} C_VEL
LIN {X 0,Y 587.331,Z 208.823,A -85,B 0,C 180,E1 -1319.83,E2 -1319.83} C_VEL
LIN {X 0,Y 587.349,Z 208.817,A -85,B 0,C 180,E1 -1322.307,E2 -1322.307} C_VEL
LIN {X 0,Y 587.332,Z 208.819,A -85,B 0,C 180,E1 -1324.483,E2 -1324.483} C_VEL
LIN {X 0,Y 587.338,Z 208.828,A -85,B 0,C 180,E1 -1327.486,E2 -1327.486} C_VEL
LIN {X 0,Y 587.34,Z 208.818,A -85,B 0,C 180,E1 -1330.425,E2 -1330.425} C_VEL
LIN {X 0,Y 587.349,Z 208.827,A -85,B 0,C 180,E1 -1333.311,E2 -1333.311} C_VEL
LIN {X 0,Y 587.356,Z 208.816,A -85,B 0,C 180,E1 -1336.154,E2 -1336.154} C_VEL
LIN {X 0,Y 587.341,Z 208.824,A -85,B 0,C 180,E1 -1338.962,E2 -1338.962} C_VEL
LIN {X 0,Y 587.367,Z 208.817,A -85,B 0,C 180,E1 -1341.745,E2 -1341.745} C_VEL
LIN {X 0,Y 587.362,Z 208.817,A -85,B 0,C 180,E1 -1344.507,E2 -1344.507} C_VEL
LIN {X 0,Y 587.37,Z 208.821,A -85,B 0,C 180,E1 -1347.257,E2 -1347.257} C_VEL
LIN {X 0,Y 587.382,Z 208.813,A -85,B 0,C 180,E1 -1350,E2 -1350} C_VEL
LIN {X 0,Y 587.37,Z 208.821,A -85,B 0,C 180,E1 -1352.743,E2 -1352.743} C_VEL
LIN {X 0,Y 587.362,Z 208.817,A -85,B 0,C 180,E1 -1355.493,E2 -1355.493} C_VEL
LIN {X 0,Y 587.367,Z 208.817,A -85,B 0,C 180,E1 -1358.255,E2 -1358.255} C_VEL
LIN {X 0,Y 587.345,Z 208.822,A -85,B 0,C 180,E1 -1361.134,E2 -1361.134} C_VEL
LIN {X 0,Y 587.362,Z 208.819,A -85,B 0,C 180,E1 -1364.261,E2 -1364.261} C_VEL
LIN {X 0,Y 587.347,Z 208.818,A -85,B 0,C 180,E1 -1367.406,E2 -1367.406} C_VEL
LIN {X 0,Y 587.328,Z 208.825,A -85,B 0,C 180,E1 -1370.305,E2 -1370.305} C_VEL
LIN {X 0,Y 587.319,Z 208.821,A -85,B 0,C 180,E1 -1373.259,E2 -1373.259} C_VEL
LIN {X 0,Y 587.332,Z 208.819,A -85,B 0,C 180,E1 -1375.517,E2 -1375.517} C_VEL
LIN {X 0,Y 587.347,Z 208.819,A -85,B 0,C 180,E1 -1377.818,E2 -1377.818} C_VEL
LIN {X 0,Y 587.338,Z 208.826,A -85,B 0,C 180,E1 -1380.511,E2 -1380.511} C_VEL
LIN {X 0,Y 587.337,Z 208.818,A -85,B 0,C 180,E1 -1383.112,E2 -1383.112} C_VEL
LIN {X 0,Y 587.308,Z 208.824,A -85,B 0,C 180,E1 -1385.899,E2 -1385.899} C_VEL
LIN {X 0,Y 587.331,Z 208.825,A -85,B 0,C 180,E1 -1388.479,E2 -1388.479} C_VEL
LIN {X 0,Y 587.334,Z 208.816,A -85,B 0,C 180,E1 -1391.157,E2 -1391.157} C_VEL
LIN {X 0,Y 587.331,Z 208.827,A -85,B 0,C 180,E1 -1394.114,E2 -1394.114} C_VEL
LIN {X 0,Y 587.318,Z 208.82,A -85,B 0,C 180,E1 -1396.994,E2 -1396.994} C_VEL
LIN {X 0,Y 587.317,Z 208.825,A -85,B 0,C 180,E1 -1399.746,E2 -1399.746} C_VEL
LIN {X 0,Y 587.344,Z 208.821,A -85,B 0,C 180,E1 -1402.393,E2 -1402.393} C_VEL
LIN {X 0,Y 587.322,Z 208.819,A -85,B 0,C 180,E1 -1404.945,E2 -1404.945} C_VEL
LIN {X 0,Y 587.336,Z 208.821,A -85,B 0,C 180,E1 -1407.421,E2 -1407.421} C_VEL
LIN {X 0,Y 587.333,Z 208.828,A -85,B 0,C 180,E1 -1409.83,E2 -1409.83} C_VEL
LIN {X 0,Y 587.348,Z 208.816,A -85,B 0,C 180,E1 -1412.307,E2 -1412.307} C_VEL
LIN {X 0,Y 587.332,Z 208.819,A -85,B 0,C 180,E1 -1414.484,E2 -1414.484} C_VEL
LIN {X 0,Y 587.316,Z 208.823,A -85,B 0,C 180,E1 -1417.132,E2 -1417.132} C_VEL
LIN {X 0,Y 587.328,Z 208.826,A -85,B 0,C 180,E1 -1419.696,E2 -1419.696} C_VEL
LIN {X 0,Y 587.347,Z 208.816,A -85,B 0,C 180,E1 -1422.594,E2 -1422.594} C_VEL
LIN {X 0,Y 587.363,Z 208.82,A -85,B 0,C 180,E1 -1425.74,E2 -1425.74} C_VEL
LIN {X 0,Y 587.347,Z 208.818,A -85,B 0,C 180,E1 -1428.867,E2 -1428.867} C_VEL
LIN {X 0,Y 587.371,Z 208.817,A -85,B 0,C 180,E1 -1431.745,E2 -1431.745} C_VEL
LIN {X 0,Y 587.355,Z 208.816,A -85,B 0,C 180,E1 -1434.507,E2 -1434.507} C_VEL
LIN {X 0,Y 587.373,Z 208.822,A -85,B 0,C 180,E1 -1437.257,E2 -1437.257} C_VEL
LIN {X 0,Y 587.383,Z 208.81,A -85,B 0,C 180,E1 -1440,E2 -1440} C_VEL
LIN {X 0,Y 587.363,Z 208.818,A -85,B 0,C 180,E1 -1442.744,E2 -1442.744} C_VEL
LIN {X 0,Y 587.365,Z 208.818,A -85,B 0,C 180,E1 -1445.493,E2 -1445.493} C_VEL
LIN {X 0,Y 587.341,Z 208.816,A -85,B 0,C 180,E1 -1448.256,E2 -1448.256} C_VEL
LIN {X 0,Y 587.348,Z 208.823,A -85,B 0,C 180,E1 -1451.134,E2 -1451.134} C_VEL
LIN {X 0,Y 587.364,Z 208.816,A -85,B 0,C 180,E1 -1454.26,E2 -1454.26} C_VEL
LIN {X 0,Y 587.343,Z 208.817,A -85,B 0,C 180,E1 -1457.407,E2 -1457.407} C_VEL
LIN {X 0,Y 587.325,Z 208.821,A -85,B 0,C 180,E1 -1460.305,E2 -1460.305} C_VEL
LIN {X 0,Y 587.32,Z 208.822,A -85,B 0,C 180,E1 -1463.259,E2 -1463.259} C_VEL
LIN {X 0,Y 587.33,Z 208.818,A -85,B 0,C 180,E1 -1465.517,E2 -1465.517} C_VEL
LIN {X 0,Y 587.347,Z 208.816,A -85,B 0,C 180,E1 -1467.818,E2 -1467.818} C_VEL
LIN {X 0,Y 587.326,Z 208.828,A -85,B 0,C 180,E1 -1470.508,E2 -1470.508} C_VEL
LIN {X 0,Y 587.338,Z 208.818,A -85,B 0,C 180,E1 -1473.112,E2 -1473.112} C_VEL
LIN {X 0,Y 587.29,Z 208.825,A -85,B 0,C 180,E1 -1475.9,E2 -1475.9} C_VEL
LIN {X 0,Y 587.328,Z 208.828,A -85,B 0,C 180,E1 -1478.48,E2 -1478.48} C_VEL
LIN {X 0,Y 587.335,Z 208.819,A -85,B 0,C 180,E1 -1481.157,E2 -1481.157} C_VEL
LIN {X 0,Y 587.328,Z 208.826,A -85,B 0,C 180,E1 -1484.114,E2 -1484.114} C_VEL
LIN {X 0,Y 587.313,Z 208.822,A -85,B 0,C 180,E1 -1486.994,E2 -1486.994} C_VEL
LIN {X 0,Y 587.315,Z 208.822,A -85,B 0,C 180,E1 -1489.746,E2 -1489.746} C_VEL
LIN {X 0,Y 587.345,Z 208.823,A -85,B 0,C 180,E1 -1492.393,E2 -1492.393} C_VEL
LIN {X 0,Y 587.344,Z 208.82,A -85,B 0,C 180,E1 -1495.653,E2 -1495.653} C_VEL
LIN {X 0,Y 587.338,Z 208.826,A -85,B 0,C 180,E1 -1498.231,E2 -1498.231} C_VEL
LIN {X 0,Y 587.347,Z 208.818,A -85,B 0,C 180,E1 -1500.868,E2 -1500.868} C_VEL
LIN {X 0,Y 587.311,Z 208.83,A -85,B 0,C 180,E1 -1503.72,E2 -1503.72} C_VEL
LIN {X 0,Y 587.355,Z 209.008,A -85,B 0,C 180,E1 -1505.42,E2 -1505.42} C_VEL
LIN {X 0,Y 587.704,Z 214.214,A -85,B 0,C 180,E1 -1506.384,E2 -1506.384} C_VEL
LIN {X 0,Y 587.574,Z 230.81,A -85,B 0,C 180,E1 -1509.338,E2 -1509.338} C_VEL
LIN {X 0,Y 587.488,Z 246.332,A -85,B 0,C 180,E1 -1512.059,E2 -1512.059} C_VEL
LIN {X 0,Y 587.372,Z 262.889,A -85,B 0,C 180,E1 -1514.916,E2 -1514.916} C_VEL
LIN {X 0,Y 587.387,Z 272.235,A -85,B 0,C 180,E1 -1516.486,E2 -1516.486} C_VEL
LIN {X 0,Y 587.709,Z 274.724,A -85,B 0,C 180,E1 -1516.559,E2 -1516.559} C_VEL
LIN {X 0,Y 587.728,Z 378.767,A -85,B 0,C 180,E1 -1517.855,E2 -1517.855} C_VEL
LIN {X 0,Y 587.68,Z 391.499,A -85,B 0,C 180,E1 -1518.139,E2 -1518.139} C_VEL
LIN {X 0,Y 587.609,Z 404.822,A -85,B 0,C 180,E1 -1518.592,E2 -1518.592} C_VEL
LIN {X 0,Y 587.555,Z 416.564,A -85,B 0,C 180,E1 -1519.141,E2 -1519.141} C_VEL
LIN {X 0,Y 587.443,Z 426.88,A -85,B 0,C 180,E1 -1519.749,E2 -1519.749} C_VEL
LIN {X 0,Y 587.381,Z 437.547,A -85,B 0,C 180,E1 -1520.531,E2 -1520.531} C_VEL
LIN {X 0,Y 587.322,Z 447.12,A -85,B 0,C 180,E1 -1521.398,E2 -1521.398} C_VEL
LIN {X 0,Y 587.273,Z 454.937,A -85,B 0,C 180,E1 -1522.263,E2 -1522.263} C_VEL
LIN {X 0,Y 587.229,Z 461.45,A -85,B 0,C 180,E1 -1523.126,E2 -1523.126} C_VEL
LIN {X 0,Y 587.23,Z 467.834,A -85,B 0,C 180,E1 -1524.161,E2 -1524.161} C_VEL
LIN {X 0,Y 587.146,Z 472.93,A -85,B 0,C 180,E1 -1525.194,E2 -1525.194} C_VEL
LIN {X 0,Y 587.213,Z 476.88,A -85,B 0,C 180,E1 -1526.226,E2 -1526.226} C_VEL
LIN {X 0,Y 587.132,Z 479.793,A -85,B 0,C 180,E1 -1527.256,E2 -1527.256} C_VEL
LIN {X 0,Y 587.147,Z 482.189,A -85,B 0,C 180,E1 -1528.628,E2 -1528.628} C_VEL
LIN {X 0,Y 587.14,Z 482.782,A -85,B 0,C 180,E1 -1529.314,E2 -1529.314} C_VEL
LIN {X 0,Y 587.14,Z 482.782,A -85,B 0,C 180,E1 -1530.686,E2 -1530.686} C_VEL
LIN {X 0,Y 587.147,Z 482.189,A -85,B 0,C 180,E1 -1531.372,E2 -1531.372} C_VEL
LIN {X 0,Y 587.132,Z 479.793,A -85,B 0,C 180,E1 -1532.744,E2 -1532.744} C_VEL
LIN {X 0,Y 587.213,Z 476.88,A -85,B 0,C 180,E1 -1533.774,E2 -1533.774} C_VEL
LIN {X 0,Y 587.146,Z 472.93,A -85,B 0,C 180,E1 -1534.806,E2 -1534.806} C_VEL
LIN {X 0,Y 587.23,Z 467.834,A -85,B 0,C 180,E1 -1535.839,E2 -1535.839} C_VEL
LIN {X 0,Y 587.229,Z 461.45,A -85,B 0,C 180,E1 -1536.874,E2 -1536.874} C_VEL
LIN {X 0,Y 587.288,Z 453.49,A -85,B 0,C 180,E1 -1537.91,E2 -1537.91} C_VEL
LIN {X 0,Y 587.335,Z 445.349,A -85,B 0,C 180,E1 -1538.776,E2 -1538.776} C_VEL
LIN {X 0,Y 587.389,Z 435.353,A -85,B 0,C 180,E1 -1539.643,E2 -1539.643} C_VEL
LIN {X 0,Y 587.466,Z 425.531,A -85,B 0,C 180,E1 -1540.338,E2 -1540.338} C_VEL
LIN {X 0,Y 587.552,Z 414.931,A -85,B 0,C 180,E1 -1540.946,E2 -1540.946} C_VEL
LIN {X 0,Y 587.616,Z 401.237,A -85,B 0,C 180,E1 -1541.547,E2 -1541.547} C_VEL
LIN {X 0,Y 587.718,Z 388.959,A -85,B 0,C 180,E1 -1541.926,E2 -1541.926} C_VEL
LIN {X 0,Y 587.733,Z 377.436,A -85,B 0,C 180,E1 -1542.167,E2 -1542.167} C_VEL
LIN {X 0,Y 587.726,Z 274.724,A -85,B 0,C 180,E1 -1543.44,E2 -1543.44} C_VEL
LIN {X 0,Y 587.387,Z 272.236,A -85,B 0,C 180,E1 -1543.514,E2 -1543.514} C_VEL
LIN {X 0,Y 587.441,Z 256.68,A -85,B 0,C 180,E1 -1546.15,E2 -1546.15} C_VEL
LIN {X 0,Y 587.52,Z 241.158,A -85,B 0,C 180,E1 -1548.843,E2 -1548.843} C_VEL
LIN {X 0,Y 587.636,Z 225.637,A -85,B 0,C 180,E1 -1551.577,E2 -1551.577} C_VEL
LIN {X 0,Y 587.729,Z 212.126,A -85,B 0,C 180,E1 -1553.989,E2 -1553.989} C_VEL
LIN {X 0,Y 587.362,Z 208.88,A -85,B 0,C 180,E1 -1554.629,E2 -1554.629} C_VEL
LIN {X 0,Y 587.34,Z 208.826,A -85,B 0,C 180,E1 -1557.818,E2 -1557.818} C_VEL
LIN {X 0,Y 587.337,Z 208.821,A -85,B 0,C 180,E1 -1560.509,E2 -1560.509} C_VEL
LIN {X 0,Y 587.335,Z 208.821,A -85,B 0,C 180,E1 -1563.396,E2 -1563.396} C_VEL
LIN {X 0,Y 587.291,Z 208.833,A -85,B 0,C 180,E1 -1565.9,E2 -1565.9} C_VEL
LIN {X 0,Y 587.326,Z 208.821,A -85,B 0,C 180,E1 -1568.479,E2 -1568.479} C_VEL
LIN {X 0,Y 587.336,Z 208.818,A -85,B 0,C 180,E1 -1571.157,E2 -1571.157} C_VEL
LIN {X 0,Y 587.313,Z 208.825,A -85,B 0,C 180,E1 -1574.112,E2 -1574.112} C_VEL
LIN {X 0,Y 587.318,Z 208.821,A -85,B 0,C 180,E1 -1576.993,E2 -1576.993} C_VEL
LIN {X 0,Y 587.312,Z 208.828,A -85,B 0,C 180,E1 -1579.745,E2 -1579.745} C_VEL
LIN {X 0,Y 587.344,Z 208.817,A -85,B 0,C 180,E1 -1582.392,E2 -1582.392} C_VEL
LIN {X 0,Y 587.343,Z 208.823,A -85,B 0,C 180,E1 -1585.653,E2 -1585.653} C_VEL
LIN {X 0,Y 587.34,Z 208.818,A -85,B 0,C 180,E1 -1588.231,E2 -1588.231} C_VEL
LIN {X 0,Y 587.349,Z 208.819,A -85,B 0,C 180,E1 -1590.866,E2 -1590.866} C_VEL
LIN {X 0,Y 587.337,Z 208.821,A -85,B 0,C 180,E1 -1593.721,E2 -1593.721} C_VEL
LIN {X 0,Y 587.323,Z 208.82,A -85,B 0,C 180,E1 -1595.993,E2 -1595.993} C_VEL
LIN {X 0,Y 587.318,Z 208.82,A -85,B 0,C 180,E1 -1598.225,E2 -1598.225} C_VEL
LIN {X 0,Y 587.346,Z 208.824,A -85,B 0,C 180,E1 -1601.151,E2 -1601.151} C_VEL
LIN {X 0,Y 587.319,Z 208.82,A -85,B 0,C 180,E1 -1604.024,E2 -1604.024} C_VEL
LIN {X 0,Y 587.357,Z 208.815,A -85,B 0,C 180,E1 -1606.154,E2 -1606.154} C_VEL
LIN {X 0,Y 587.338,Z 208.826,A -85,B 0,C 180,E1 -1608.962,E2 -1608.962} C_VEL
LIN {X 0,Y 587.341,Z 208.816,A -85,B 0,C 180,E1 -1611.744,E2 -1611.744} C_VEL
LIN {X 0,Y 587.365,Z 208.818,A -85,B 0,C 180,E1 -1614.507,E2 -1614.507} C_VEL
LIN {X 0,Y 587.363,Z 208.818,A -85,B 0,C 180,E1 -1617.256,E2 -1617.256} C_VEL
LIN {X 0,Y 587.383,Z 208.81,A -85,B 0,C 180,E1 -1620,E2 -1620} C_VEL
LIN {X 0,Y 587.373,Z 208.822,A -85,B 0,C 180,E1 -1622.743,E2 -1622.743} C_VEL
LIN {X 0,Y 587.356,Z 208.816,A -85,B 0,C 180,E1 -1625.493,E2 -1625.493} C_VEL
LIN {X 0,Y 587.371,Z 208.817,A -85,B 0,C 180,E1 -1628.255,E2 -1628.255} C_VEL
LIN {X 0,Y 587.347,Z 208.818,A -85,B 0,C 180,E1 -1631.133,E2 -1631.133} C_VEL
LIN {X 0,Y 587.363,Z 208.82,A -85,B 0,C 180,E1 -1634.26,E2 -1634.26} C_VEL
LIN {X 0,Y 587.347,Z 208.816,A -85,B 0,C 180,E1 -1637.406,E2 -1637.406} C_VEL
LIN {X 0,Y 587.308,Z 208.824,A -85,B 0,C 180,E1 -1638.314,E2 -1638.314} C_VEL
LIN {X 0,Y 586.665,Z 208.903,A -85,B 0,C 180,E1 -1638.886,E2 -1638.886} C_VEL
LIN {X 0,Y 583.839,Z 209.253,A -85,B 0,C 180,E1 -1639.814,E2 -1639.814} C_VEL
LIN {X 0,Y 581.428,Z 209.561,A -85,B 0,C 180,E1 -1640.562,E2 -1640.562} C_VEL
LIN {X 0,Y 580.376,Z 209.686,A -85,B 0,C 180,E1 -1641.138,E2 -1641.138} C_VEL
LIN {X 0,Y 580.281,Z 209.696,A -85,B 0,C 180,E1 -1641.333,E2 -1641.333} C_VEL
LIN {X 0,Y 580.296,Z 209.705,A -85,B 0,C 180,E1 -1644.316,E2 -1644.316} C_VEL
LIN {X 0,Y 580.275,Z 209.699,A -85,B 0,C 180,E1 -1646.623,E2 -1646.623} C_VEL
LIN {X 0,Y 580.299,Z 209.694,A -85,B 0,C 180,E1 -1649.31,E2 -1649.31} C_VEL
LIN {X 0,Y 580.299,Z 209.704,A -85,B 0,C 180,E1 -1652.2,E2 -1652.2} C_VEL
LIN {X 0,Y 580.287,Z 209.697,A -85,B 0,C 180,E1 -1654.696,E2 -1654.696} C_VEL
LIN {X 0,Y 580.298,Z 209.695,A -85,B 0,C 180,E1 -1657.268,E2 -1657.268} C_VEL
LIN {X 0,Y 580.295,Z 209.699,A -85,B 0,C 180,E1 -1660.271,E2 -1660.271} C_VEL
LIN {X 0,Y 580.278,Z 209.698,A -85,B 0,C 180,E1 -1662.706,E2 -1662.706} C_VEL
LIN {X 0,Y 580.271,Z 209.703,A -85,B 0,C 180,E1 -1665.608,E2 -1665.608} C_VEL
LIN {X 0,Y 580.311,Z 209.694,A -85,B 0,C 180,E1 -1668.234,E2 -1668.234} C_VEL
LIN {X 0,Y 580.287,Z 209.696,A -85,B 0,C 180,E1 -1670.966,E2 -1670.966} C_VEL
LIN {X 0,Y 580.276,Z 209.706,A -85,B 0,C 180,E1 -1673.597,E2 -1673.597} C_VEL
LIN {X 0,Y 580.313,Z 209.695,A -85,B 0,C 180,E1 -1676.145,E2 -1676.145} C_VEL
LIN {X 0,Y 580.285,Z 209.697,A -85,B 0,C 180,E1 -1678.615,E2 -1678.615} C_VEL
LIN {X 0,Y 580.292,Z 209.696,A -85,B 0,C 180,E1 -1681.024,E2 -1681.024} C_VEL
LIN {X 0,Y 580.289,Z 209.704,A -85,B 0,C 180,E1 -1683.666,E2 -1683.666} C_VEL
LIN {X 0,Y 580.297,Z 209.702,A -85,B 0,C 180,E1 -1685.684,E2 -1685.684} C_VEL
LIN {X 0,Y 580.271,Z 209.701,A -85,B 0,C 180,E1 -1687.947,E2 -1687.947} C_VEL
LIN {X 0,Y 580.316,Z 209.696,A -85,B 0,C 180,E1 -1690.914,E2 -1690.914} C_VEL
LIN {X 0,Y 580.276,Z 209.701,A -85,B 0,C 180,E1 -1693.826,E2 -1693.826} C_VEL
LIN {X 0,Y 580.323,Z 209.693,A -85,B 0,C 180,E1 -1695.983,E2 -1695.983} C_VEL
LIN {X 0,Y 580.301,Z 209.699,A -85,B 0,C 180,E1 -1698.827,E2 -1698.827} C_VEL
LIN {X 0,Y 580.331,Z 209.695,A -85,B 0,C 180,E1 -1701.644,E2 -1701.644} C_VEL
LIN {X 0,Y 580.329,Z 209.693,A -85,B 0,C 180,E1 -1704.44,E2 -1704.44} C_VEL
LIN {X 0,Y 580.344,Z 209.69,A -85,B 0,C 180,E1 -1707.918,E2 -1707.918} C_VEL
LIN {X 0,Y 580.359,Z 209.694,A -85,B 0,C 180,E1 -1710.694,E2 -1710.694} C_VEL
LIN {X 0,Y 580.281,Z 209.7,A -85,B 0,C 180,E1 -1713.472,E2 -1713.472} C_VEL
LIN {X 0,Y 580.329,Z 209.693,A -85,B 0,C 180,E1 -1715.56,E2 -1715.56} C_VEL
LIN {X 0,Y 580.331,Z 209.695,A -85,B 0,C 180,E1 -1718.356,E2 -1718.356} C_VEL
LIN {X 0,Y 580.297,Z 209.699,A -85,B 0,C 180,E1 -1721.191,E2 -1721.191} C_VEL
LIN {X 0,Y 580.323,Z 209.693,A -85,B 0,C 180,E1 -1724.017,E2 -1724.017} C_VEL
LIN {X 0,Y 580.309,Z 209.7,A -85,B 0,C 180,E1 -1726.914,E2 -1726.914} C_VEL
LIN {X 0,Y 580.303,Z 209.695,A -85,B 0,C 180,E1 -1729.822,E2 -1729.822} C_VEL
LIN {X 0,Y 580.292,Z 209.702,A -85,B 0,C 180,E1 -1732.802,E2 -1732.802} C_VEL
LIN {X 0,Y 580.304,Z 209.696,A -85,B 0,C 180,E1 -1735.08,E2 -1735.08} C_VEL
LIN {X 0,Y 580.3,Z 209.701,A -85,B 0,C 180,E1 -1738.185,E2 -1738.185} C_VEL
LIN {X 0,Y 580.289,Z 209.701,A -85,B 0,C 180,E1 -1740.696,E2 -1740.696} C_VEL
LIN {X 0,Y 580.301,Z 209.694,A -85,B 0,C 180,E1 -1743.317,E2 -1743.317} C_VEL
LIN {X 0,Y 580.266,Z 209.699,A -85,B 0,C 180,E1 -1745.76,E2 -1745.76} C_VEL
LIN {X 0,Y 580.287,Z 209.705,A -85,B 0,C 180,E1 -1748.146,E2 -1748.146} C_VEL
LIN {X 0,Y 580.298,Z 209.693,A -85,B 0,C 180,E1 -1750.843,E2 -1750.843} C_VEL
LIN {X 0,Y 580.285,Z 209.696,A -85,B 0,C 180,E1 -1753.657,E2 -1753.657} C_VEL
LIN {X 0,Y 580.282,Z 209.699,A -85,B 0,C 180,E1 -1756.609,E2 -1756.609} C_VEL
LIN {X 0,Y 580.298,Z 209.694,A -85,B 0,C 180,E1 -1759.157,E2 -1759.157} C_VEL
LIN {X 0,Y 580.288,Z 209.706,A -85,B 0,C 180,E1 -1761.927,E2 -1761.927} C_VEL
LIN {X 0,Y 580.282,Z 209.698,A -85,B 0,C 180,E1 -1764.455,E2 -1764.455} C_VEL
LIN {X 0,Y 580.288,Z 209.695,A -85,B 0,C 180,E1 -1766.976,E2 -1766.976} C_VEL
LIN {X 0,Y 580.3,Z 209.699,A -85,B 0,C 180,E1 -1769.426,E2 -1769.426} C_VEL
LIN {X 0,Y 580.295,Z 209.696,A -85,B 0,C 180,E1 -1772.142,E2 -1772.142} C_VEL
LIN {X 0,Y 580.319,Z 209.695,A -85,B 0,C 180,E1 -1775.27,E2 -1775.27} C_VEL
LIN {X 0,Y 580.273,Z 209.702,A -85,B 0,C 180,E1 -1777.948,E2 -1777.948} C_VEL
LIN {X 0,Y 580.317,Z 209.691,A -85,B 0,C 180,E1 -1780.914,E2 -1780.914} C_VEL
LIN {X 0,Y 580.277,Z 209.702,A -85,B 0,C 180,E1 -1783.826,E2 -1783.826} C_VEL
LIN {X 0,Y 580.323,Z 209.694,A -85,B 0,C 180,E1 -1785.983,E2 -1785.983} C_VEL
LIN {X 0,Y 580.303,Z 209.694,A -85,B 0,C 180,E1 -1788.827,E2 -1788.827} C_VEL
LIN {X 0,Y 580.334,Z 209.695,A -85,B 0,C 180,E1 -1791.644,E2 -1791.644} C_VEL
LIN {X 0,Y 580.324,Z 209.692,A -85,B 0,C 180,E1 -1794.441,E2 -1794.441} C_VEL
LIN {X 0,Y 580.346,Z 209.688,A -85,B 0,C 180,E1 -1797.918,E2 -1797.918} C_VEL
LIN {X 0,Y 580.354,Z 209.687,A -85,B 0,C 180,E1 -1800.694,E2 -1800.694} C_VEL
LIN {X 0,Y 580.288,Z 209.701,A -85,B 0,C 180,E1 -1803.472,E2 -1803.472} C_VEL
LIN {X 0,Y 580.331,Z 209.693,A -85,B 0,C 180,E1 -1805.56,E2 -1805.56} C_VEL
LIN {X 0,Y 580.31,Z 209.693,A -85,B 0,C 180,E1 -1808.357,E2 -1808.357} C_VEL
LIN {X 0,Y 580.3,Z 209.7,A -85,B 0,C 180,E1 -1811.191,E2 -1811.191} C_VEL
LIN {X 0,Y 580.325,Z 209.691,A -85,B 0,C 180,E1 -1814.017,E2 -1814.017} C_VEL
LIN {X 0,Y 580.313,Z 209.7,A -85,B 0,C 180,E1 -1816.914,E2 -1816.914} C_VEL
LIN {X 0,Y 580.286,Z 209.694,A -85,B 0,C 180,E1 -1819.823,E2 -1819.823} C_VEL
LIN {X 0,Y 580.269,Z 209.699,A -85,B 0,C 180,E1 -1822.053,E2 -1822.053} C_VEL
LIN {X 0,Y 580.305,Z 209.696,A -85,B 0,C 180,E1 -1825.08,E2 -1825.08} C_VEL
LIN {X 0,Y 580.299,Z 209.696,A -85,B 0,C 180,E1 -1828.186,E2 -1828.186} C_VEL
LIN {X 0,Y 580.277,Z 209.706,A -85,B 0,C 180,E1 -1830.694,E2 -1830.694} C_VEL
LIN {X 0,Y 580.284,Z 209.695,A -85,B 0,C 180,E1 -1833.314,E2 -1833.314} C_VEL
LIN {X 0,Y 580.245,Z 209.702,A -85,B 0,C 180,E1 -1835.756,E2 -1835.756} C_VEL
LIN {X 0,Y 580.287,Z 209.702,A -85,B 0,C 180,E1 -1838.147,E2 -1838.147} C_VEL
LIN {X 0,Y 580.298,Z 209.698,A -85,B 0,C 180,E1 -1840.844,E2 -1840.844} C_VEL
LIN {X 0,Y 580.28,Z 209.698,A -85,B 0,C 180,E1 -1843.658,E2 -1843.658} C_VEL
LIN {X 0,Y 580.275,Z 209.702,A -85,B 0,C 180,E1 -1846.61,E2 -1846.61} C_VEL
LIN {X 0,Y 580.299,Z 209.692,A -85,B 0,C 180,E1 -1849.157,E2 -1849.157} C_VEL
LIN {X 0,Y 580.289,Z 209.702,A -85,B 0,C 180,E1 -1851.928,E2 -1851.928} C_VEL
LIN {X 0,Y 580.252,Z 209.705,A -85,B 0,C 180,E1 -1854.453,E2 -1854.453} C_VEL
LIN {X 0,Y 580.29,Z 209.696,A -85,B 0,C 180,E1 -1856.975,E2 -1856.975} C_VEL
LIN {X 0,Y 580.296,Z 209.698,A -85,B 0,C 180,E1 -1859.425,E2 -1859.425} C_VEL
LIN {X 0,Y 580.291,Z 209.705,A -85,B 0,C 180,E1 -1862.143,E2 -1862.143} C_VEL
LIN {X 0,Y 580.286,Z 209.779,A -85,B 0,C 180,E1 -1865.243,E2 -1865.243} C_VEL
LIN {X 0,Y 580.765,Z 214.098,A -85,B 0,C 180,E1 -1866.084,E2 -1866.084} C_VEL
LIN {X 0,Y 580.596,Z 230.953,A -85,B 0,C 180,E1 -1869.104,E2 -1869.104} C_VEL
LIN {X 0,Y 580.469,Z 245.298,A -85,B 0,C 180,E1 -1871.652,E2 -1871.652} C_VEL
LIN {X 0,Y 580.403,Z 260.819,A -85,B 0,C 180,E1 -1874.37,E2 -1874.37} C_VEL
LIN {X 0,Y 580.342,Z 272.243,A -85,B 0,C 180,E1 -1876.318,E2 -1876.318} C_VEL
LIN {X 0,Y 580.678,Z 274.724,A -85,B 0,C 180,E1 -1876.393,E2 -1876.393} C_VEL
LIN {X 0,Y 580.945,Z 283.667,A -85,B 0,C 180,E1 -1876.511,E2 -1876.511} C_VEL
LIN {X 0,Y 580.81,Z 378.707,A -85,B 0,C 180,E1 -1877.708,E2 -1877.708} C_VEL
LIN {X 0,Y 580.734,Z 391.506,A -85,B 0,C 180,E1 -1877.995,E2 -1877.995} C_VEL
LIN {X 0,Y 580.636,Z 405.428,A -85,B 0,C 180,E1 -1878.48,E2 -1878.48} C_VEL
LIN {X 0,Y 580.567,Z 416.544,A -85,B 0,C 180,E1 -1879.009,E2 -1879.009} C_VEL
LIN {X 0,Y 580.45,Z 426.862,A -85,B 0,C 180,E1 -1879.624,E2 -1879.624} C_VEL
LIN {X 0,Y 580.361,Z 437.551,A -85,B 0,C 180,E1 -1880.415,E2 -1880.415} C_VEL
LIN {X 0,Y 580.271,Z 447.118,A -85,B 0,C 180,E1 -1881.292,E2 -1881.292} C_VEL
LIN {X 0,Y 580.221,Z 454.928,A -85,B 0,C 180,E1 -1882.168,E2 -1882.168} C_VEL
LIN {X 0,Y 580.157,Z 461.44,A -85,B 0,C 180,E1 -1883.042,E2 -1883.042} C_VEL
LIN {X 0,Y 580.162,Z 467.824,A -85,B 0,C 180,E1 -1884.09,E2 -1884.09} C_VEL
LIN {X 0,Y 580.053,Z 472.92,A -85,B 0,C 180,E1 -1885.135,E2 -1885.135} C_VEL
LIN {X 0,Y 580.11,Z 476.872,A -85,B 0,C 180,E1 -1886.179,E2 -1886.179} C_VEL
LIN {X 0,Y 580.043,Z 479.787,A -85,B 0,C 180,E1 -1887.222,E2 -1887.222} C_VEL
LIN {X 0,Y 580.047,Z 482.191,A -85,B 0,C 180,E1 -1888.611,E2 -1888.611} C_VEL
LIN {X 0,Y 580.04,Z 482.781,A -85,B 0,C 180,E1 -1889.306,E2 -1889.306} C_VEL
LIN {X 0,Y 580.04,Z 482.781,A -85,B 0,C 180,E1 -1890.694,E2 -1890.694} C_VEL
LIN {X 0,Y 580.047,Z 482.191,A -85,B 0,C 180,E1 -1891.389,E2 -1891.389} C_VEL
LIN {X 0,Y 580.043,Z 479.787,A -85,B 0,C 180,E1 -1892.778,E2 -1892.778} C_VEL
LIN {X 0,Y 580.11,Z 476.872,A -85,B 0,C 180,E1 -1893.821,E2 -1893.821} C_VEL
LIN {X 0,Y 580.053,Z 472.92,A -85,B 0,C 180,E1 -1894.865,E2 -1894.865} C_VEL
LIN {X 0,Y 580.162,Z 467.824,A -85,B 0,C 180,E1 -1895.91,E2 -1895.91} C_VEL
LIN {X 0,Y 580.157,Z 461.44,A -85,B 0,C 180,E1 -1896.958,E2 -1896.958} C_VEL
LIN {X 0,Y 580.242,Z 453.494,A -85,B 0,C 180,E1 -1898.007,E2 -1898.007} C_VEL
LIN {X 0,Y 580.304,Z 445.353,A -85,B 0,C 180,E1 -1898.883,E2 -1898.883} C_VEL
LIN {X 0,Y 580.357,Z 435.338,A -85,B 0,C 180,E1 -1899.761,E2 -1899.761} C_VEL
LIN {X 0,Y 580.463,Z 425.514,A -85,B 0,C 180,E1 -1900.464,E2 -1900.464} C_VEL
LIN {X 0,Y 580.578,Z 414.915,A -85,B 0,C 180,E1 -1901.079,E2 -1901.079} C_VEL
LIN {X 0,Y 580.658,Z 402.161,A -85,B 0,C 180,E1 -1901.652,E2 -1901.652} C_VEL
LIN {X 0,Y 580.775,Z 389.796,A -85,B 0,C 180,E1 -1902.049,E2 -1902.049} C_VEL
LIN {X 0,Y 580.81,Z 378.707,A -85,B 0,C 180,E1 -1902.292,E2 -1902.292} C_VEL
LIN {X 0,Y 580.817,Z 275.395,A -85,B 0,C 180,E1 -1903.595,E2 -1903.595} C_VEL
LIN {X 0,Y 580.386,Z 272.559,A -85,B 0,C 180,E1 -1903.658,E2 -1903.658} C_VEL
LIN {X 0,Y 580.326,Z 270.133,A -85,B 0,C 180,E1 -1904.017,E2 -1904.017} C_VEL
LIN {X 0,Y 580.4,Z 254.611,A -85,B 0,C 180,E1 -1906.713,E2 -1906.713} C_VEL
LIN {X 0,Y 580.547,Z 240.354,A -85,B 0,C 180,E1 -1909.221,E2 -1909.221} C_VEL
LIN {X 0,Y 580.667,Z 225.605,A -85,B 0,C 180,E1 -1911.85,E2 -1911.85} C_VEL
LIN {X 0,Y 580.751,Z 213.076,A -85,B 0,C 180,E1 -1914.106,E2 -1914.106} C_VEL
LIN {X 0,Y 580.286,Z 209.778,A -85,B 0,C 180,E1 -1914.757,E2 -1914.757} C_VEL
LIN {X 0,Y 580.291,Z 209.705,A -85,B 0,C 180,E1 -1917.857,E2 -1917.857} C_VEL
LIN {X 0,Y 580.285,Z 209.699,A -85,B 0,C 180,E1 -1920.694,E2 -1920.694} C_VEL
LIN {X 0,Y 580.304,Z 209.696,A -85,B 0,C 180,E1 -1923.316,E2 -1923.316} C_VEL
LIN {X 0,Y 580.246,Z 209.709,A -85,B 0,C 180,E1 -1925.756,E2 -1925.756} C_VEL
LIN {X 0,Y 580.287,Z 209.701,A -85,B 0,C 180,E1 -1928.146,E2 -1928.146} C_VEL
LIN {X 0,Y 580.299,Z 209.692,A -85,B 0,C 180,E1 -1930.843,E2 -1930.843} C_VEL
LIN {X 0,Y 580.274,Z 209.707,A -85,B 0,C 180,E1 -1933.658,E2 -1933.658} C_VEL
LIN {X 0,Y 580.279,Z 209.697,A -85,B 0,C 180,E1 -1936.609,E2 -1936.609} C_VEL
LIN {X 0,Y 580.298,Z 209.698,A -85,B 0,C 180,E1 -1939.156,E2 -1939.156} C_VEL
LIN {X 0,Y 580.289,Z 209.7,A -85,B 0,C 180,E1 -1941.927,E2 -1941.927} C_VEL
LIN {X 0,Y 580.25,Z 209.7,A -85,B 0,C 180,E1 -1944.452,E2 -1944.452} C_VEL
LIN {X 0,Y 580.29,Z 209.697,A -85,B 0,C 180,E1 -1946.975,E2 -1946.975} C_VEL
LIN {X 0,Y 580.287,Z 209.706,A -85,B 0,C 180,E1 -1949.424,E2 -1949.424} C_VEL
LIN {X 0,Y 580.298,Z 209.693,A -85,B 0,C 180,E1 -1952.141,E2 -1952.141} C_VEL
LIN {X 0,Y 580.321,Z 209.7,A -85,B 0,C 180,E1 -1955.27,E2 -1955.27} C_VEL
LIN {X 0,Y 580.269,Z 209.699,A -85,B 0,C 180,E1 -1957.947,E2 -1957.947} C_VEL
LIN {X 0,Y 580.298,Z 209.698,A -85,B 0,C 180,E1 -1960.913,E2 -1960.913} C_VEL
LIN {X 0,Y 580.273,Z 209.698,A -85,B 0,C 180,E1 -1963.825,E2 -1963.825} C_VEL
LIN {X 0,Y 580.325,Z 209.691,A -85,B 0,C 180,E1 -1965.983,E2 -1965.983} C_VEL
LIN {X 0,Y 580.305,Z 209.7,A -85,B 0,C 180,E1 -1968.827,E2 -1968.827} C_VEL
LIN {X 0,Y 580.31,Z 209.693,A -85,B 0,C 180,E1 -1971.643,E2 -1971.643} C_VEL
LIN {X 0,Y 580.331,Z 209.693,A -85,B 0,C 180,E1 -1974.44,E2 -1974.44} C_VEL
LIN {X 0,Y 580.331,Z 209.694,A -85,B 0,C 180,E1 -1977.223,E2 -1977.223} C_VEL
LIN {X 0,Y 580.352,Z 209.685,A -85,B 0,C 180,E1 -1980,E2 -1980} C_VEL
LIN {X 0,Y 580.339,Z 209.699,A -85,B 0,C 180,E1 -1982.776,E2 -1982.776} C_VEL
LIN {X 0,Y 580.324,Z 209.692,A -85,B 0,C 180,E1 -1985.559,E2 -1985.559} C_VEL
LIN {X 0,Y 580.334,Z 209.695,A -85,B 0,C 180,E1 -1988.356,E2 -1988.356} C_VEL
LIN {X 0,Y 580.299,Z 209.695,A -85,B 0,C 180,E1 -1991.191,E2 -1991.191} C_VEL
LIN {X 0,Y 580.323,Z 209.694,A -85,B 0,C 180,E1 -1994.017,E2 -1994.017} C_VEL
LIN {X 0,Y 580.31,Z 209.695,A -85,B 0,C 180,E1 -1996.913,E2 -1996.913} C_VEL
LIN {X 0,Y 580.303,Z 209.693,A -85,B 0,C 180,E1 -1999.822,E2 -1999.822} C_VEL
LIN {X 0,Y 580.281,Z 209.696,A -85,B 0,C 180,E1 -2001.333,E2 -2001.333} C_VEL
LIN {X 0,Y 579.585,Z 209.787,A -85,B 0,C 180,E1 -2001.912,E2 -2001.912} C_VEL
LIN {X 0,Y 576.706,Z 210.145,A -85,B 0,C 180,E1 -2002.852,E2 -2002.852} C_VEL
LIN {X 0,Y 574.31,Z 210.443,A -85,B 0,C 180,E1 -2003.608,E2 -2003.608} C_VEL
LIN {X 0,Y 573.312,Z 210.573,A -85,B 0,C 180,E1 -2004.192,E2 -2004.192} C_VEL
LIN {X 0,Y 573.246,Z 210.576,A -85,B 0,C 180,E1 -2004.39,E2 -2004.39} C_VEL
LIN {X 0,Y 573.248,Z 210.571,A -85,B 0,C 180,E1 -2006.976,E2 -2006.976} C_VEL
LIN {X 0,Y 573.245,Z 210.574,A -85,B 0,C 180,E1 -2009.488,E2 -2009.488} C_VEL
LIN {X 0,Y 573.252,Z 210.581,A -85,B 0,C 180,E1 -2012.229,E2 -2012.229} C_VEL
LIN {X 0,Y 573.236,Z 210.574,A -85,B 0,C 180,E1 -2014.772,E2 -2014.772} C_VEL
LIN {X 0,Y 573.252,Z 210.573,A -85,B 0,C 180,E1 -2017.166,E2 -2017.166} C_VEL
LIN {X 0,Y 573.245,Z 210.577,A -85,B 0,C 180,E1 -2019.607,E2 -2019.607} C_VEL
LIN {X 0,Y 573.24,Z 210.575,A -85,B 0,C 180,E1 -2022.642,E2 -2022.642} C_VEL
LIN {X 0,Y 573.236,Z 210.58,A -85,B 0,C 180,E1 -2025.667,E2 -2025.667} C_VEL
LIN {X 0,Y 573.241,Z 210.571,A -85,B 0,C 180,E1 -2028.544,E2 -2028.544} C_VEL
LIN {X 0,Y 573.246,Z 210.576,A -85,B 0,C 180,E1 -2031.299,E2 -2031.299} C_VEL
LIN {X 0,Y 573.239,Z 210.577,A -85,B 0,C 180,E1 -2034.014,E2 -2034.014} C_VEL
LIN {X 0,Y 573.282,Z 210.568,A -85,B 0,C 180,E1 -2036.519,E2 -2036.519} C_VEL
LIN {X 0,Y 573.235,Z 210.578,A -85,B 0,C 180,E1 -2039.116,E2 -2039.116} C_VEL
LIN {X 0,Y 573.262,Z 210.576,A -85,B 0,C 180,E1 -2041.968,E2 -2041.968} C_VEL
LIN {X 0,Y 573.251,Z 210.573,A -85,B 0,C 180,E1 -2044.59,E2 -2044.59} C_VEL
LIN {X 0,Y 573.235,Z 210.582,A -85,B 0,C 180,E1 -2047.662,E2 -2047.662} C_VEL
LIN {X 0,Y 573.275,Z 210.572,A -85,B 0,C 180,E1 -2050.728,E2 -2050.728} C_VEL
LIN {X 0,Y 573.248,Z 210.579,A -85,B 0,C 180,E1 -2053.622,E2 -2053.622} C_VEL
LIN {X 0,Y 573.27,Z 210.574,A -85,B 0,C 180,E1 -2055.807,E2 -2055.807} C_VEL
LIN {X 0,Y 573.26,Z 210.576,A -85,B 0,C 180,E1 -2058.745,E2 -2058.745} C_VEL
LIN {X 0,Y 573.287,Z 210.574,A -85,B 0,C 180,E1 -2061.541,E2 -2061.541} C_VEL
LIN {X 0,Y 573.297,Z 210.569,A -85,B 0,C 180,E1 -2064.372,E2 -2064.372} C_VEL
LIN {X 0,Y 573.314,Z 210.566,A -85,B 0,C 180,E1 -2067.892,E2 -2067.892} C_VEL
LIN {X 0,Y 573.329,Z 210.57,A -85,B 0,C 180,E1 -2070.702,E2 -2070.702} C_VEL
LIN {X 0,Y 573.303,Z 210.575,A -85,B 0,C 180,E1 -2072.811,E2 -2072.811} C_VEL
LIN {X 0,Y 573.297,Z 210.569,A -85,B 0,C 180,E1 -2075.628,E2 -2075.628} C_VEL
LIN {X 0,Y 573.287,Z 210.574,A -85,B 0,C 180,E1 -2078.459,E2 -2078.459} C_VEL
LIN {X 0,Y 573.268,Z 210.574,A -85,B 0,C 180,E1 -2081.312,E2 -2081.312} C_VEL
LIN {X 0,Y 573.27,Z 210.574,A -85,B 0,C 180,E1 -2084.193,E2 -2084.193} C_VEL
LIN {X 0,Y 573.255,Z 210.576,A -85,B 0,C 180,E1 -2087.112,E2 -2087.112} C_VEL
LIN {X 0,Y 573.25,Z 210.576,A -85,B 0,C 180,E1 -2090.077,E2 -2090.077} C_VEL
LIN {X 0,Y 573.231,Z 210.578,A -85,B 0,C 180,E1 -2093.099,E2 -2093.099} C_VEL
LIN {X 0,Y 573.252,Z 210.573,A -85,B 0,C 180,E1 -2095.41,E2 -2095.41} C_VEL
LIN {X 0,Y 573.262,Z 210.576,A -85,B 0,C 180,E1 -2098.032,E2 -2098.032} C_VEL
LIN {X 0,Y 573.235,Z 210.578,A -85,B 0,C 180,E1 -2100.884,E2 -2100.884} C_VEL
LIN {X 0,Y 573.258,Z 210.571,A -85,B 0,C 180,E1 -2103.524,E2 -2103.524} C_VEL
LIN {X 0,Y 573.239,Z 210.578,A -85,B 0,C 180,E1 -2106.05,E2 -2106.05} C_VEL
LIN {X 0,Y 573.246,Z 210.576,A -85,B 0,C 180,E1 -2108.701,E2 -2108.701} C_VEL
LIN {X 0,Y 573.25,Z 210.571,A -85,B 0,C 180,E1 -2111.596,E2 -2111.596} C_VEL
LIN {X 0,Y 573.236,Z 210.58,A -85,B 0,C 180,E1 -2114.333,E2 -2114.333} C_VEL
LIN {X 0,Y 573.24,Z 210.575,A -85,B 0,C 180,E1 -2117.358,E2 -2117.358} C_VEL
LIN {X 0,Y 573.245,Z 210.577,A -85,B 0,C 180,E1 -2120.393,E2 -2120.393} C_VEL
LIN {X 0,Y 573.253,Z 210.573,A -85,B 0,C 180,E1 -2123.078,E2 -2123.078} C_VEL
LIN {X 0,Y 573.264,Z 210.576,A -85,B 0,C 180,E1 -2125.672,E2 -2125.672} C_VEL
LIN {X 0,Y 573.246,Z 210.578,A -85,B 0,C 180,E1 -2128.185,E2 -2128.185} C_VEL
LIN {X 0,Y 573.262,Z 210.571,A -85,B 0,C 180,E1 -2130.635,E2 -2130.635} C_VEL
LIN {X 0,Y 573.248,Z 210.571,A -85,B 0,C 180,E1 -2133.024,E2 -2133.024} C_VEL
LIN {X 0,Y 573.273,Z 210.574,A -85,B 0,C 180,E1 -2135.366,E2 -2135.366} C_VEL
LIN {X 0,Y 573.228,Z 210.575,A -85,B 0,C 180,E1 -2138.42,E2 -2138.42} C_VEL
LIN {X 0,Y 573.277,Z 210.566,A -85,B 0,C 180,E1 -2140.729,E2 -2140.729} C_VEL
LIN {X 0,Y 573.25,Z 210.581,A -85,B 0,C 180,E1 -2143.622,E2 -2143.622} C_VEL
LIN {X 0,Y 573.271,Z 210.575,A -85,B 0,C 180,E1 -2145.807,E2 -2145.807} C_VEL
LIN {X 0,Y 573.261,Z 210.57,A -85,B 0,C 180,E1 -2148.745,E2 -2148.745} C_VEL
LIN {X 0,Y 573.289,Z 210.574,A -85,B 0,C 180,E1 -2151.541,E2 -2151.541} C_VEL
LIN {X 0,Y 573.293,Z 210.568,A -85,B 0,C 180,E1 -2154.372,E2 -2154.372} C_VEL
LIN {X 0,Y 573.316,Z 210.564,A -85,B 0,C 180,E1 -2157.893,E2 -2157.893} C_VEL
LIN {X 0,Y 573.325,Z 210.562,A -85,B 0,C 180,E1 -2160.703,E2 -2160.703} C_VEL
LIN {X 0,Y 573.299,Z 210.57,A -85,B 0,C 180,E1 -2162.811,E2 -2162.811} C_VEL
LIN {X 0,Y 573.297,Z 210.569,A -85,B 0,C 180,E1 -2165.628,E2 -2165.628} C_VEL
LIN {X 0,Y 573.255,Z 210.572,A -85,B 0,C 180,E1 -2168.46,E2 -2168.46} C_VEL
LIN {X 0,Y 573.272,Z 210.573,A -85,B 0,C 180,E1 -2171.312,E2 -2171.312} C_VEL
LIN {X 0,Y 573.281,Z 210.571,A -85,B 0,C 180,E1 -2174.425,E2 -2174.425} C_VEL
LIN {X 0,Y 573.258,Z 210.574,A -85,B 0,C 180,E1 -2177.112,E2 -2177.112} C_VEL
LIN {X 0,Y 573.241,Z 210.572,A -85,B 0,C 180,E1 -2180.077,E2 -2180.077} C_VEL
LIN {X 0,Y 573.235,Z 210.578,A -85,B 0,C 180,E1 -2182.338,E2 -2182.338} C_VEL
LIN {X 0,Y 573.249,Z 210.572,A -85,B 0,C 180,E1 -2185.411,E2 -2185.411} C_VEL
LIN {X 0,Y 573.251,Z 210.572,A -85,B 0,C 180,E1 -2188.029,E2 -2188.029} C_VEL
LIN {X 0,Y 573.224,Z 210.581,A -85,B 0,C 180,E1 -2190.882,E2 -2190.882} C_VEL
LIN {X 0,Y 573.241,Z 210.572,A -85,B 0,C 180,E1 -2193.521,E2 -2193.521} C_VEL
LIN {X 0,Y 573.215,Z 210.58,A -85,B 0,C 180,E1 -2196.052,E2 -2196.052} C_VEL
LIN {X 0,Y 573.242,Z 210.578,A -85,B 0,C 180,E1 -2198.702,E2 -2198.702} C_VEL
LIN {X 0,Y 573.231,Z 210.576,A -85,B 0,C 180,E1 -2201.593,E2 -2201.593} C_VEL
LIN {X 0,Y 573.234,Z 210.584,A -85,B 0,C 180,E1 -2204.334,E2 -2204.334} C_VEL
LIN {X 0,Y 573.241,Z 210.574,A -85,B 0,C 180,E1 -2207.359,E2 -2207.359} C_VEL
LIN {X 0,Y 573.248,Z 210.58,A -85,B 0,C 180,E1 -2210.393,E2 -2210.393} C_VEL
LIN {X 0,Y 573.253,Z 210.572,A -85,B 0,C 180,E1 -2213.078,E2 -2213.078} C_VEL
LIN {X 0,Y 573.266,Z 210.574,A -85,B 0,C 180,E1 -2215.671,E2 -2215.671} C_VEL
LIN {X 0,Y 573.239,Z 210.583,A -85,B 0,C 180,E1 -2218.185,E2 -2218.185} C_VEL
LIN {X 0,Y 573.262,Z 210.574,A -85,B 0,C 180,E1 -2220.634,E2 -2220.634} C_VEL
LIN {X 0,Y 573.211,Z 210.58,A -85,B 0,C 180,E1 -2223.022,E2 -2223.022} C_VEL
LIN {X 0,Y 573.263,Z 210.711,A -85,B 0,C 180,E1 -2225.124,E2 -2225.124} C_VEL
LIN {X 0,Y 573.821,Z 215.048,A -85,B 0,C 180,E1 -2225.969,E2 -2225.969} C_VEL
LIN {X 0,Y 573.602,Z 231.195,A -85,B 0,C 180,E1 -2228.899,E2 -2228.899} C_VEL
LIN {X 0,Y 573.518,Z 244.263,A -85,B 0,C 180,E1 -2231.236,E2 -2231.236} C_VEL
LIN {X 0,Y 573.403,Z 258.75,A -85,B 0,C 180,E1 -2233.809,E2 -2233.809} C_VEL
LIN {X 0,Y 573.308,Z 272.252,A -85,B 0,C 180,E1 -2236.147,E2 -2236.147} C_VEL
LIN {X 0,Y 573.623,Z 274.429,A -85,B 0,C 180,E1 -2236.219,E2 -2236.219} C_VEL
LIN {X 0,Y 574.044,Z 280.09,A -85,B 0,C 180,E1 -2236.301,E2 -2236.301} C_VEL
LIN {X 0,Y 573.888,Z 378.646,A -85,B 0,C 180,E1 -2237.558,E2 -2237.558} C_VEL
LIN {X 0,Y 573.837,Z 390.633,A -85,B 0,C 180,E1 -2237.826,E2 -2237.826} C_VEL
LIN {X 0,Y 573.701,Z 404.394,A -85,B 0,C 180,E1 -2238.294,E2 -2238.294} C_VEL
LIN {X 0,Y 573.596,Z 415.374,A -85,B 0,C 180,E1 -2238.81,E2 -2238.81} C_VEL
LIN {X 0,Y 573.467,Z 425.496,A -85,B 0,C 180,E1 -2239.407,E2 -2239.407} C_VEL
LIN {X 0,Y 573.338,Z 435.324,A -85,B 0,C 180,E1 -2240.118,E2 -2240.118} C_VEL
LIN {X 0,Y 573.279,Z 445.356,A -85,B 0,C 180,E1 -2241.007,E2 -2241.007} C_VEL
LIN {X 0,Y 573.161,Z 454.918,A -85,B 0,C 180,E1 -2242.071,E2 -2242.071} C_VEL
LIN {X 0,Y 573.082,Z 461.43,A -85,B 0,C 180,E1 -2242.956,E2 -2242.956} C_VEL
LIN {X 0,Y 573.074,Z 467.814,A -85,B 0,C 180,E1 -2244.017,E2 -2244.017} C_VEL
LIN {X 0,Y 572.962,Z 472.911,A -85,B 0,C 180,E1 -2245.074,E2 -2245.074} C_VEL
LIN {X 0,Y 573.015,Z 476.864,A -85,B 0,C 180,E1 -2246.132,E2 -2246.132} C_VEL
LIN {X 0,Y 572.959,Z 479.782,A -85,B 0,C 180,E1 -2247.188,E2 -2247.188} C_VEL
LIN {X 0,Y 572.946,Z 482.193,A -85,B 0,C 180,E1 -2248.594,E2 -2248.594} C_VEL
LIN {X 0,Y 572.941,Z 482.781,A -85,B 0,C 180,E1 -2249.297,E2 -2249.297} C_VEL
LIN {X 0,Y 572.941,Z 482.781,A -85,B 0,C 180,E1 -2250.703,E2 -2250.703} C_VEL
LIN {X 0,Y 572.946,Z 482.193,A -85,B 0,C 180,E1 -2251.406,E2 -2251.406} C_VEL
LIN {X 0,Y 572.959,Z 479.782,A -85,B 0,C 180,E1 -2252.812,E2 -2252.812} C_VEL
LIN {X 0,Y 573.015,Z 476.864,A -85,B 0,C 180,E1 -2253.868,E2 -2253.868} C_VEL
LIN {X 0,Y 572.962,Z 472.911,A -85,B 0,C 180,E1 -2254.926,E2 -2254.926} C_VEL
LIN {X 0,Y 573.074,Z 467.814,A -85,B 0,C 180,E1 -2255.983,E2 -2255.983} C_VEL
LIN {X 0,Y 573.082,Z 461.43,A -85,B 0,C 180,E1 -2257.044,E2 -2257.044} C_VEL
LIN {X 0,Y 573.177,Z 453.498,A -85,B 0,C 180,E1 -2258.106,E2 -2258.106} C_VEL
LIN {X 0,Y 573.279,Z 445.356,A -85,B 0,C 180,E1 -2258.993,E2 -2258.993} C_VEL
LIN {X 0,Y 573.338,Z 435.324,A -85,B 0,C 180,E1 -2259.882,E2 -2259.882} C_VEL
LIN {X 0,Y 573.467,Z 425.496,A -85,B 0,C 180,E1 -2260.593,E2 -2260.593} C_VEL
LIN {X 0,Y 573.622,Z 414.294,A -85,B 0,C 180,E1 -2261.248,E2 -2261.248} C_VEL
LIN {X 0,Y 573.705,Z 400.928,A -85,B 0,C 180,E1 -2261.84,E2 -2261.84} C_VEL
LIN {X 0,Y 573.834,Z 388.885,A -85,B 0,C 180,E1 -2262.219,E2 -2262.219} C_VEL
LIN {X 0,Y 573.888,Z 378.646,A -85,B 0,C 180,E1 -2262.442,E2 -2262.442} C_VEL
LIN {X 0,Y 573.942,Z 276.413,A -85,B 0,C 180,E1 -2263.748,E2 -2263.748} C_VEL
LIN {X 0,Y 573.346,Z 272.572,A -85,B 0,C 180,E1 -2263.829,E2 -2263.829} C_VEL
LIN {X 0,Y 573.287,Z 270.133,A -85,B 0,C 180,E1 -2264.193,E2 -2264.193} C_VEL
LIN {X 0,Y 573.388,Z 255.797,A -85,B 0,C 180,E1 -2266.714,E2 -2266.714} C_VEL
LIN {X 0,Y 573.565,Z 242.193,A -85,B 0,C 180,E1 -2269.134,E2 -2269.134} C_VEL
LIN {X 0,Y 573.687,Z 227.565,A -85,B 0,C 180,E1 -2271.751,E2 -2271.751} C_VEL
LIN {X 0,Y 573.788,Z 214.026,A -85,B 0,C 180,E1 -2274.225,E2 -2274.225} C_VEL
LIN {X 0,Y 573.261,Z 210.626,A -85,B 0,C 180,E1 -2274.912,E2 -2274.912} C_VEL
LIN {X 0,Y 573.246,Z 210.582,A -85,B 0,C 180,E1 -2278.027,E2 -2278.027} C_VEL
LIN {X 0,Y 573.247,Z 210.582,A -85,B 0,C 180,E1 -2280.176,E2 -2280.176} C_VEL
LIN {X 0,Y 573.254,Z 210.574,A -85,B 0,C 180,E1 -2282.645,E2 -2282.645} C_VEL
LIN {X 0,Y 573.207,Z 210.579,A -85,B 0,C 180,E1 -2285.188,E2 -2285.188} C_VEL
LIN {X 0,Y 573.236,Z 210.584,A -85,B 0,C 180,E1 -2287.807,E2 -2287.807} C_VEL
LIN {X 0,Y 573.246,Z 210.571,A -85,B 0,C 180,E1 -2290.525,E2 -2290.525} C_VEL
LIN {X 0,Y 573.237,Z 210.579,A -85,B 0,C 180,E1 -2293.359,E2 -2293.359} C_VEL
LIN {X 0,Y 573.246,Z 210.575,A -85,B 0,C 180,E1 -2296.331,E2 -2296.331} C_VEL
LIN {X 0,Y 573.23,Z 210.575,A -85,B 0,C 180,E1 -2298.543,E2 -2298.543} C_VEL
LIN {X 0,Y 573.242,Z 210.578,A -85,B 0,C 180,E1 -2301.298,E2 -2301.298} C_VEL
LIN {X 0,Y 573.213,Z 210.579,A -85,B 0,C 180,E1 -2304.018,E2 -2304.018} C_VEL
LIN {X 0,Y 573.239,Z 210.572,A -85,B 0,C 180,E1 -2306.515,E2 -2306.515} C_VEL
LIN {X 0,Y 573.224,Z 210.581,A -85,B 0,C 180,E1 -2309.118,E2 -2309.118} C_VEL
LIN {X 0,Y 573.251,Z 210.572,A -85,B 0,C 180,E1 -2311.971,E2 -2311.971} C_VEL
LIN {X 0,Y 573.249,Z 210.572,A -85,B 0,C 180,E1 -2314.589,E2 -2314.589} C_VEL
LIN {X 0,Y 573.235,Z 210.578,A -85,B 0,C 180,E1 -2317.662,E2 -2317.662} C_VEL
LIN {X 0,Y 573.266,Z 210.571,A -85,B 0,C 180,E1 -2320.67,E2 -2320.67} C_VEL
LIN {X 0,Y 573.245,Z 210.575,A -85,B 0,C 180,E1 -2323.621,E2 -2323.621} C_VEL
LIN {X 0,Y 573.272,Z 210.571,A -85,B 0,C 180,E1 -2325.807,E2 -2325.807} C_VEL
LIN {X 0,Y 573.263,Z 210.575,A -85,B 0,C 180,E1 -2328.745,E2 -2328.745} C_VEL
LIN {X 0,Y 573.255,Z 210.572,A -85,B 0,C 180,E1 -2331.54,E2 -2331.54} C_VEL
LIN {X 0,Y 573.297,Z 210.569,A -85,B 0,C 180,E1 -2334.372,E2 -2334.372} C_VEL
LIN {X 0,Y 573.313,Z 210.564,A -85,B 0,C 180,E1 -2337.892,E2 -2337.892} C_VEL
LIN {X 0,Y 573.335,Z 210.567,A -85,B 0,C 180,E1 -2340.702,E2 -2340.702} C_VEL
LIN {X 0,Y 573.305,Z 210.575,A -85,B 0,C 180,E1 -2342.81,E2 -2342.81} C_VEL
LIN {X 0,Y 573.293,Z 210.568,A -85,B 0,C 180,E1 -2345.628,E2 -2345.628} C_VEL
LIN {X 0,Y 573.289,Z 210.574,A -85,B 0,C 180,E1 -2348.459,E2 -2348.459} C_VEL
LIN {X 0,Y 573.27,Z 210.569,A -85,B 0,C 180,E1 -2351.312,E2 -2351.312} C_VEL
LIN {X 0,Y 573.28,Z 210.578,A -85,B 0,C 180,E1 -2354.424,E2 -2354.424} C_VEL
LIN {X 0,Y 573.256,Z 210.572,A -85,B 0,C 180,E1 -2357.111,E2 -2357.111} C_VEL
LIN {X 0,Y 573.251,Z 210.574,A -85,B 0,C 180,E1 -2360.076,E2 -2360.076} C_VEL
LIN {X 0,Y 573.232,Z 210.576,A -85,B 0,C 180,E1 -2363.099,E2 -2363.099} C_VEL
LIN {X 0,Y 573.246,Z 210.576,A -85,B 0,C 180,E1 -2364.39,E2 -2364.39} C_VEL
LIN {X 0,Y 572.622,Z 210.655,A -85,B 0,C 180,E1 -2364.976,E2 -2364.976} C_VEL
LIN {X 0,Y 569.78,Z 211.009,A -85,B 0,C 180,E1 -2365.927,E2 -2365.927} C_VEL
LIN {X 0,Y 567.346,Z 211.308,A -85,B 0,C 180,E1 -2366.693,E2 -2366.693} C_VEL
LIN {X 0,Y 566.29,Z 211.436,A -85,B 0,C 180,E1 -2367.284,E2 -2367.284} C_VEL
LIN {X 0,Y 566.2,Z 211.448,A -85,B 0,C 180,E1 -2367.484,E2 -2367.484} C_VEL
LIN {X 0,Y 566.199,Z 211.454,A -85,B 0,C 180,E1 -2369.768,E2 -2369.768} C_VEL
LIN {X 0,Y 566.204,Z 211.455,A -85,B 0,C 180,E1 -2372.43,E2 -2372.43} C_VEL
LIN {X 0,Y 566.198,Z 211.449,A -85,B 0,C 180,E1 -2374.992,E2 -2374.992} C_VEL
LIN {X 0,Y 566.194,Z 211.454,A -85,B 0,C 180,E1 -2377.46,E2 -2377.46} C_VEL
LIN {X 0,Y 566.224,Z 211.453,A -85,B 0,C 180,E1 -2380.197,E2 -2380.197} C_VEL
LIN {X 0,Y 566.202,Z 211.451,A -85,B 0,C 180,E1 -2383.053,E2 -2383.053} C_VEL
LIN {X 0,Y 566.199,Z 211.454,A -85,B 0,C 180,E1 -2386.048,E2 -2386.048} C_VEL
LIN {X 0,Y 566.208,Z 211.445,A -85,B 0,C 180,E1 -2388.864,E2 -2388.864} C_VEL
LIN {X 0,Y 566.187,Z 211.46,A -85,B 0,C 180,E1 -2391.637,E2 -2391.637} C_VEL
LIN {X 0,Y 566.19,Z 211.451,A -85,B 0,C 180,E1 -2394.31,E2 -2394.31} C_VEL
LIN {X 0,Y 566.226,Z 211.447,A -85,B 0,C 180,E1 -2396.898,E2 -2396.898} C_VEL
LIN {X 0,Y 566.185,Z 211.46,A -85,B 0,C 180,E1 -2399.408,E2 -2399.408} C_VEL
LIN {X 0,Y 566.225,Z 211.454,A -85,B 0,C 180,E1 -2401.858,E2 -2401.858} C_VEL
LIN {X 0,Y 566.211,Z 211.451,A -85,B 0,C 180,E1 -2404.251,E2 -2404.251} C_VEL
LIN {X 0,Y 566.17,Z 211.456,A -85,B 0,C 180,E1 -2406.718,E2 -2406.718} C_VEL
LIN {X 0,Y 566.211,Z 211.456,A -85,B 0,C 180,E1 -2409.663,E2 -2409.663} C_VEL
LIN {X 0,Y 566.197,Z 211.454,A -85,B 0,C 180,E1 -2412.668,E2 -2412.668} C_VEL
LIN {X 0,Y 566.231,Z 211.453,A -85,B 0,C 180,E1 -2415.627,E2 -2415.627} C_VEL
LIN {X 0,Y 566.232,Z 211.451,A -85,B 0,C 180,E1 -2418.675,E2 -2418.675} C_VEL
LIN {X 0,Y 566.231,Z 211.454,A -85,B 0,C 180,E1 -2421.434,E2 -2421.434} C_VEL
LIN {X 0,Y 566.266,Z 211.444,A -85,B 0,C 180,E1 -2424.302,E2 -2424.302} C_VEL
LIN {X 0,Y 566.284,Z 211.442,A -85,B 0,C 180,E1 -2427.866,E2 -2427.866} C_VEL
LIN {X 0,Y 566.3,Z 211.446,A -85,B 0,C 180,E1 -2430.711,E2 -2430.711} C_VEL
LIN {X 0,Y 566.269,Z 211.452,A -85,B 0,C 180,E1 -2432.846,E2 -2432.846} C_VEL
LIN {X 0,Y 566.266,Z 211.444,A -85,B 0,C 180,E1 -2435.698,E2 -2435.698} C_VEL
LIN {X 0,Y 566.231,Z 211.454,A -85,B 0,C 180,E1 -2438.566,E2 -2438.566} C_VEL
LIN {X 0,Y 566.239,Z 211.449,A -85,B 0,C 180,E1 -2441.454,E2 -2441.454} C_VEL
LIN {X 0,Y 566.231,Z 211.455,A -85,B 0,C 180,E1 -2444.507,E2 -2444.507} C_VEL
LIN {X 0,Y 566.197,Z 211.454,A -85,B 0,C 180,E1 -2447.332,E2 -2447.332} C_VEL
LIN {X 0,Y 566.211,Z 211.456,A -85,B 0,C 180,E1 -2450.337,E2 -2450.337} C_VEL
LIN {X 0,Y 566.169,Z 211.456,A -85,B 0,C 180,E1 -2453.282,E2 -2453.282} C_VEL
LIN {X 0,Y 566.212,Z 211.451,A -85,B 0,C 180,E1 -2455.749,E2 -2455.749} C_VEL
LIN {X 0,Y 566.204,Z 211.457,A -85,B 0,C 180,E1 -2458.203,E2 -2458.203} C_VEL
LIN {X 0,Y 566.196,Z 211.453,A -85,B 0,C 180,E1 -2461.078,E2 -2461.078} C_VEL
LIN {X 0,Y 566.208,Z 211.451,A -85,B 0,C 180,E1 -2463.734,E2 -2463.734} C_VEL
LIN {X 0,Y 566.207,Z 211.456,A -85,B 0,C 180,E1 -2466.569,E2 -2466.569} C_VEL
LIN {X 0,Y 566.21,Z 211.452,A -85,B 0,C 180,E1 -2469.686,E2 -2469.686} C_VEL
LIN {X 0,Y 566.211,Z 211.452,A -85,B 0,C 180,E1 -2472.087,E2 -2472.087} C_VEL
LIN {X 0,Y 566.171,Z 211.454,A -85,B 0,C 180,E1 -2475.036,E2 -2475.036} C_VEL
LIN {X 0,Y 566.215,Z 211.456,A -85,B 0,C 180,E1 -2478.136,E2 -2478.136} C_VEL
LIN {X 0,Y 566.22,Z 211.449,A -85,B 0,C 180,E1 -2480.727,E2 -2480.727} C_VEL
LIN {X 0,Y 566.203,Z 211.459,A -85,B 0,C 180,E1 -2483.785,E2 -2483.785} C_VEL
LIN {X 0,Y 566.226,Z 211.447,A -85,B 0,C 180,E1 -2486.899,E2 -2486.899} C_VEL
LIN {X 0,Y 566.185,Z 211.457,A -85,B 0,C 180,E1 -2489.408,E2 -2489.408} C_VEL
LIN {X 0,Y 566.209,Z 211.454,A -85,B 0,C 180,E1 -2491.858,E2 -2491.858} C_VEL
LIN {X 0,Y 566.212,Z 211.451,A -85,B 0,C 180,E1 -2494.251,E2 -2494.251} C_VEL
LIN {X 0,Y 566.171,Z 211.455,A -85,B 0,C 180,E1 -2496.718,E2 -2496.718} C_VEL
LIN {X 0,Y 566.212,Z 211.454,A -85,B 0,C 180,E1 -2499.663,E2 -2499.663} C_VEL
LIN {X 0,Y 566.198,Z 211.45,A -85,B 0,C 180,E1 -2502.669,E2 -2502.669} C_VEL
LIN {X 0,Y 566.232,Z 211.454,A -85,B 0,C 180,E1 -2505.627,E2 -2505.627} C_VEL
LIN {X 0,Y 566.233,Z 211.445,A -85,B 0,C 180,E1 -2508.676,E2 -2508.676} C_VEL
LIN {X 0,Y 566.233,Z 211.454,A -85,B 0,C 180,E1 -2511.435,E2 -2511.435} C_VEL
LIN {X 0,Y 566.261,Z 211.443,A -85,B 0,C 180,E1 -2514.302,E2 -2514.302} C_VEL
LIN {X 0,Y 566.286,Z 211.439,A -85,B 0,C 180,E1 -2517.867,E2 -2517.867} C_VEL
LIN {X 0,Y 566.297,Z 211.437,A -85,B 0,C 180,E1 -2520.711,E2 -2520.711} C_VEL
LIN {X 0,Y 566.267,Z 211.446,A -85,B 0,C 180,E1 -2522.846,E2 -2522.846} C_VEL
LIN {X 0,Y 566.264,Z 211.444,A -85,B 0,C 180,E1 -2525.699,E2 -2525.699} C_VEL
LIN {X 0,Y 566.206,Z 211.451,A -85,B 0,C 180,E1 -2528.566,E2 -2528.566} C_VEL
LIN {X 0,Y 566.242,Z 211.447,A -85,B 0,C 180,E1 -2531.455,E2 -2531.455} C_VEL
LIN {X 0,Y 566.234,Z 211.45,A -85,B 0,C 180,E1 -2534.507,E2 -2534.507} C_VEL
LIN {X 0,Y 566.197,Z 211.451,A -85,B 0,C 180,E1 -2537.332,E2 -2537.332} C_VEL
LIN {X 0,Y 566.207,Z 211.45,A -85,B 0,C 180,E1 -2540.338,E2 -2540.338} C_VEL
LIN {X 0,Y 566.172,Z 211.456,A -85,B 0,C 180,E1 -2543.282,E2 -2543.282} C_VEL
LIN {X 0,Y 566.21,Z 211.448,A -85,B 0,C 180,E1 -2545.75,E2 -2545.75} C_VEL
LIN {X 0,Y 566.203,Z 211.451,A -85,B 0,C 180,E1 -2548.202,E2 -2548.202} C_VEL
LIN {X 0,Y 566.188,Z 211.455,A -85,B 0,C 180,E1 -2551.076,E2 -2551.076} C_VEL
LIN {X 0,Y 566.198,Z 211.45,A -85,B 0,C 180,E1 -2553.732,E2 -2553.732} C_VEL
LIN {X 0,Y 566.2,Z 211.46,A -85,B 0,C 180,E1 -2556.57,E2 -2556.57} C_VEL
LIN {X 0,Y 566.215,Z 211.449,A -85,B 0,C 180,E1 -2559.686,E2 -2559.686} C_VEL
LIN {X 0,Y 566.204,Z 211.452,A -85,B 0,C 180,E1 -2562.918,E2 -2562.918} C_VEL
LIN {X 0,Y 566.196,Z 211.458,A -85,B 0,C 180,E1 -2566.05,E2 -2566.05} C_VEL
LIN {X 0,Y 566.205,Z 211.447,A -85,B 0,C 180,E1 -2569.215,E2 -2569.215} C_VEL
LIN {X 0,Y 566.188,Z 211.455,A -85,B 0,C 180,E1 -2571.637,E2 -2571.637} C_VEL
LIN {X 0,Y 566.163,Z 211.462,A -85,B 0,C 180,E1 -2574.308,E2 -2574.308} C_VEL
LIN {X 0,Y 566.221,Z 211.449,A -85,B 0,C 180,E1 -2576.898,E2 -2576.898} C_VEL
LIN {X 0,Y 566.181,Z 211.457,A -85,B 0,C 180,E1 -2579.407,E2 -2579.407} C_VEL
LIN {X 0,Y 566.194,Z 211.461,A -85,B 0,C 180,E1 -2581.857,E2 -2581.857} C_VEL
LIN {X 0,Y 566.227,Z 211.522,A -85,B 0,C 180,E1 -2584.951,E2 -2584.951} C_VEL
LIN {X 0,Y 566.861,Z 217.035,A -85,B 0,C 180,E1 -2586.044,E2 -2586.044} C_VEL
LIN {X 0,Y 566.605,Z 232.664,A -85,B 0,C 180,E1 -2588.918,E2 -2588.918} C_VEL
LIN {X 0,Y 566.477,Z 246.262,A -85,B 0,C 180,E1 -2591.369,E2 -2591.369} C_VEL
LIN {X 0,Y 566.354,Z 260.819,A -85,B 0,C 180,E1 -2593.972,E2 -2593.972} C_VEL
LIN {X 0,Y 566.28,Z 272.26,A -85,B 0,C 180,E1 -2595.972,E2 -2595.972} C_VEL
LIN {X 0,Y 566.609,Z 274.429,A -85,B 0,C 180,E1 -2596.045,E2 -2596.045} C_VEL
LIN {X 0,Y 567.146,Z 280.09,A -85,B 0,C 180,E1 -2596.131,E2 -2596.131} C_VEL
LIN {X 0,Y 566.965,Z 378.585,A -85,B 0,C 180,E1 -2597.403,E2 -2597.403} C_VEL
LIN {X 0,Y 566.896,Z 389.722,A -85,B 0,C 180,E1 -2597.652,E2 -2597.652} C_VEL
LIN {X 0,Y 566.77,Z 402.167,A -85,B 0,C 180,E1 -2598.058,E2 -2598.058} C_VEL
LIN {X 0,Y 566.642,Z 414.908,A -85,B 0,C 180,E1 -2598.646,E2 -2598.646} C_VEL
LIN {X 0,Y 566.485,Z 425.478,A -85,B 0,C 180,E1 -2599.275,E2 -2599.275} C_VEL
LIN {X 0,Y 566.392,Z 434.178,A -85,B 0,C 180,E1 -2599.906,E2 -2599.906} C_VEL
LIN {X 0,Y 566.303,Z 441.545,A -85,B 0,C 180,E1 -2600.536,E2 -2600.536} C_VEL
LIN {X 0,Y 566.159,Z 448.733,A -85,B 0,C 180,E1 -2601.253,E2 -2601.253} C_VEL
LIN {X 0,Y 566.094,Z 456.279,A -85,B 0,C 180,E1 -2602.151,E2 -2602.151} C_VEL
LIN {X 0,Y 566.004,Z 462.685,A -85,B 0,C 180,E1 -2603.064,E2 -2603.064} C_VEL
LIN {X 0,Y 565.989,Z 467.804,A -85,B 0,C 180,E1 -2603.941,E2 -2603.941} C_VEL
LIN {X 0,Y 565.877,Z 472.901,A -85,B 0,C 180,E1 -2605.013,E2 -2605.013} C_VEL
LIN {X 0,Y 565.926,Z 476.856,A -85,B 0,C 180,E1 -2606.084,E2 -2606.084} C_VEL
LIN {X 0,Y 565.878,Z 479.776,A -85,B 0,C 180,E1 -2607.152,E2 -2607.152} C_VEL
LIN {X 0,Y 565.846,Z 482.195,A -85,B 0,C 180,E1 -2608.577,E2 -2608.577} C_VEL
LIN {X 0,Y 565.841,Z 482.78,A -85,B 0,C 180,E1 -2609.288,E2 -2609.288} C_VEL
LIN {X 0,Y 565.841,Z 482.78,A -85,B 0,C 180,E1 -2610.712,E2 -2610.712} C_VEL
LIN {X 0,Y 565.846,Z 482.195,A -85,B 0,C 180,E1 -2611.423,E2 -2611.423} C_VEL
LIN {X 0,Y 565.878,Z 479.776,A -85,B 0,C 180,E1 -2612.848,E2 -2612.848} C_VEL
LIN {X 0,Y 565.926,Z 476.856,A -85,B 0,C 180,E1 -2613.916,E2 -2613.916} C_VEL
LIN {X 0,Y 565.877,Z 472.901,A -85,B 0,C 180,E1 -2614.987,E2 -2614.987} C_VEL
LIN {X 0,Y 565.99,Z 467.804,A -85,B 0,C 180,E1 -2616.059,E2 -2616.059} C_VEL
LIN {X 0,Y 566.004,Z 462.685,A -85,B 0,C 180,E1 -2616.936,E2 -2616.936} C_VEL
LIN {X 0,Y 566.094,Z 456.279,A -85,B 0,C 180,E1 -2617.849,E2 -2617.849} C_VEL
LIN {X 0,Y 566.159,Z 448.733,A -85,B 0,C 180,E1 -2618.747,E2 -2618.747} C_VEL
LIN {X 0,Y 566.295,Z 439.621,A -85,B 0,C 180,E1 -2619.645,E2 -2619.645} C_VEL
LIN {X 0,Y 566.442,Z 428.176,A -85,B 0,C 180,E1 -2620.545,E2 -2620.545} C_VEL
LIN {X 0,Y 566.56,Z 418.777,A -85,B 0,C 180,E1 -2621.14,E2 -2621.14} C_VEL
LIN {X 0,Y 566.701,Z 408.701,A -85,B 0,C 180,E1 -2621.658,E2 -2621.658} C_VEL
LIN {X 0,Y 566.787,Z 398.33,A -85,B 0,C 180,E1 -2622.078,E2 -2622.078} C_VEL
LIN {X 0,Y 566.885,Z 387.975,A -85,B 0,C 180,E1 -2622.394,E2 -2622.394} C_VEL
LIN {X 0,Y 566.961,Z 377.254,A -85,B 0,C 180,E1 -2622.62,E2 -2622.62} C_VEL
LIN {X 0,Y 567.076,Z 277.308,A -85,B 0,C 180,E1 -2623.906,E2 -2623.906} C_VEL
LIN {X 0,Y 566.32,Z 272.585,A -85,B 0,C 180,E1 -2624.004,E2 -2624.004} C_VEL
LIN {X 0,Y 566.268,Z 271.167,A -85,B 0,C 180,E1 -2624.189,E2 -2624.189} C_VEL
LIN {X 0,Y 566.415,Z 254.411,A -85,B 0,C 180,E1 -2627.174,E2 -2627.174} C_VEL
LIN {X 0,Y 566.612,Z 237.897,A -85,B 0,C 180,E1 -2630.133,E2 -2630.133} C_VEL
LIN {X 0,Y 566.816,Z 221.219,A -85,B 0,C 180,E1 -2633.183,E2 -2633.183} C_VEL
